Yaskawa INFORM job: A_ROOF_SIDE_0617_2_PAINT_52.JBI

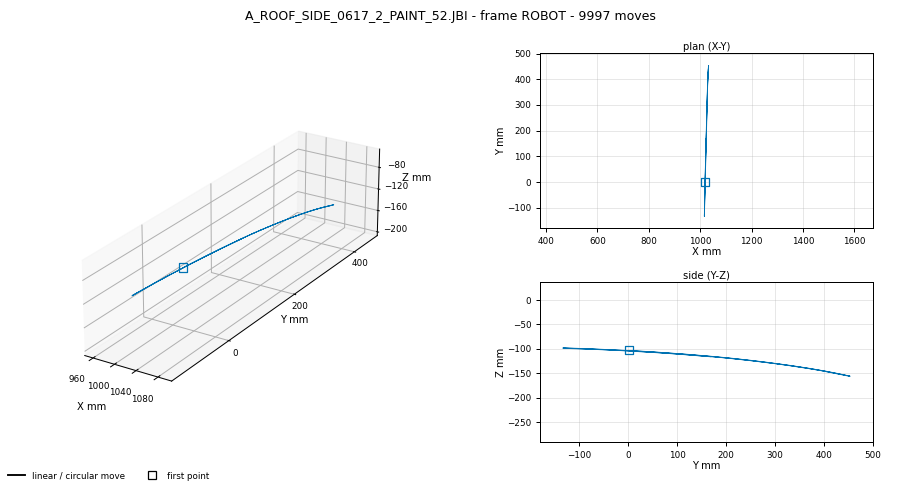
[picture p0: tool path of A_ROOF_SIDE_0617_2_PAINT_52.JBI in frame ROBOT, 9997 of 9997 moves have a stored position in this frame; points joined in program order, loops and branches not executed]
/JOB
//NAME A_ROOF_SIDE_0617_2_PAINT52
//POS
///NPOS 9997,0,0,0,0,0
///TOOL 1
///USER 0
///POSTYPE ROBOT
///RECTAN
///RCONF 1,0,0,0,0,0,0,0,0,0,0,0,0,0,0,0,0,0,0,0,0,0,0,0
C00000=1019.781,0.856,-102.921,166.512,52.317,159.512
C00001=1019.787,1.106,-102.935,166.515,52.311,159.512
C00002=1019.792,1.356,-102.949,166.518,52.306,159.511
C00003=1019.798,1.605,-102.963,166.520,52.301,159.511
C00004=1019.804,1.854,-102.976,166.523,52.295,159.510
C00005=1019.809,2.104,-102.990,166.526,52.289,159.510
C00006=1019.815,2.354,-103.004,166.529,52.284,159.509
C00007=1019.821,2.604,-103.018,166.531,52.279,159.509
C00008=1019.826,2.853,-103.032,166.533,52.273,159.508
C00009=1019.833,3.103,-103.045,166.536,52.268,159.508
C00010=1019.838,3.352,-103.059,166.540,52.262,159.507
C00011=1019.843,3.602,-103.073,166.541,52.257,159.506
C00012=1019.849,3.851,-103.087,166.544,52.251,159.506
C00013=1019.855,4.100,-103.101,166.547,52.246,159.506
C00014=1019.860,4.350,-103.115,166.550,52.240,159.505
C00015=1019.866,4.599,-103.128,166.553,52.235,159.505
C00016=1019.872,4.849,-103.142,166.555,52.230,159.504
C00017=1019.877,5.098,-103.156,166.558,52.224,159.503
C00018=1019.883,5.349,-103.170,166.561,52.218,159.503
C00019=1019.889,5.598,-103.184,166.564,52.213,159.503
C00020=1019.895,5.848,-103.197,166.565,52.207,159.502
C00021=1019.901,6.097,-103.211,166.569,52.202,159.501
C00022=1019.906,6.347,-103.225,166.572,52.197,159.501
C00023=1019.912,6.596,-103.240,166.574,52.191,159.500
C00024=1019.917,6.845,-103.254,166.577,52.186,159.500
C00025=1019.923,7.095,-103.268,166.579,52.180,159.499
C00026=1019.930,7.345,-103.281,166.582,52.175,159.499
C00027=1019.935,7.594,-103.295,166.585,52.169,159.498
C00028=1019.941,7.844,-103.309,166.588,52.163,159.498
C00029=1019.946,8.093,-103.323,166.591,52.158,159.497
C00030=1019.952,8.342,-103.337,166.594,52.152,159.497
C00031=1019.958,8.593,-103.351,166.596,52.147,159.496
C00032=1019.964,8.842,-103.365,166.598,52.141,159.496
C00033=1019.970,9.092,-103.379,166.601,52.136,159.495
C00034=1019.975,9.341,-103.392,166.604,52.130,159.495
C00035=1019.981,9.590,-103.407,166.607,52.124,159.494
C00036=1019.987,9.840,-103.421,166.609,52.119,159.493
C00037=1019.992,10.090,-103.435,166.612,52.113,159.493
C00038=1019.999,10.339,-103.448,166.614,52.107,159.492
C00039=1020.005,10.622,-103.464,166.618,52.101,159.492
C00040=1020.011,10.903,-103.481,166.621,52.095,159.491
C00041=1020.019,11.186,-103.496,166.623,52.089,159.491
C00042=1020.025,11.469,-103.512,166.627,52.083,159.490
C00043=1020.031,11.718,-103.526,166.630,52.077,159.490
C00044=1020.036,11.967,-103.541,166.633,52.071,159.489
C00045=1020.042,12.217,-103.554,166.635,52.066,159.488
C00046=1020.048,12.467,-103.569,166.637,52.060,159.488
C00047=1020.054,12.716,-103.583,166.640,52.055,159.487
C00048=1020.060,12.965,-103.597,166.643,52.049,159.487
C00049=1020.065,13.215,-103.610,166.646,52.043,159.486
C00050=1020.071,13.465,-103.625,166.649,52.037,159.486
C00051=1020.077,13.714,-103.639,166.651,52.032,159.485
C00052=1020.083,13.964,-103.653,166.654,52.026,159.485
C00053=1020.089,14.213,-103.668,166.657,52.021,159.484
C00054=1020.094,14.463,-103.682,166.660,52.016,159.484
C00055=1020.100,14.712,-103.697,166.661,52.010,159.483
C00056=1020.105,14.962,-103.711,166.664,52.005,159.483
C00057=1020.111,15.211,-103.726,166.667,51.999,159.482
C00058=1020.117,15.461,-103.740,166.670,51.994,159.482
C00059=1020.123,15.710,-103.754,166.672,51.989,159.481
C00060=1020.129,15.960,-103.769,166.675,51.983,159.480
C00061=1020.135,16.209,-103.783,166.678,51.977,159.480
C00062=1020.139,16.459,-103.798,166.681,51.971,159.479
C00063=1020.145,16.708,-103.812,166.683,51.966,159.479
C00064=1020.151,16.958,-103.826,166.685,51.960,159.478
C00065=1020.157,17.207,-103.841,166.689,51.955,159.478
C00066=1020.162,17.457,-103.855,166.691,51.949,159.477
C00067=1020.169,17.706,-103.870,166.693,51.944,159.477
C00068=1020.174,17.956,-103.884,166.696,51.938,159.476
C00069=1020.180,18.205,-103.898,166.699,51.933,159.476
C00070=1020.185,18.455,-103.913,166.702,51.927,159.475
C00071=1020.191,18.704,-103.928,166.705,51.922,159.475
C00072=1020.197,18.954,-103.941,166.707,51.916,159.474
C00073=1020.203,19.204,-103.956,166.710,51.911,159.473
C00074=1020.209,19.453,-103.971,166.713,51.906,159.473
C00075=1020.214,19.703,-103.986,166.715,51.900,159.472
C00076=1020.220,19.952,-104.000,166.717,51.895,159.472
C00077=1020.226,20.201,-104.015,166.720,51.889,159.471
C00078=1020.232,20.451,-104.029,166.723,51.883,159.471
C00079=1020.237,20.701,-104.044,166.725,51.878,159.470
C00080=1020.243,20.950,-104.059,166.728,51.873,159.470
C00081=1020.249,21.200,-104.073,166.731,51.867,159.469
C00082=1020.254,21.449,-104.088,166.734,51.861,159.469
C00083=1020.259,21.698,-104.103,166.736,51.856,159.468
C00084=1020.266,21.948,-104.117,166.739,51.850,159.467
C00085=1020.271,22.197,-104.132,166.741,51.844,159.467
C00086=1020.277,22.447,-104.147,166.744,51.839,159.466
C00087=1020.282,22.697,-104.161,166.746,51.834,159.466
C00088=1020.288,22.946,-104.176,166.749,51.828,159.465
C00089=1020.294,23.196,-104.191,166.752,51.822,159.465
C00090=1020.300,23.445,-104.206,166.755,51.817,159.464
C00091=1020.306,23.695,-104.220,166.758,51.811,159.463
C00092=1020.312,23.944,-104.235,166.760,51.806,159.463
C00093=1020.317,24.194,-104.250,166.762,51.800,159.462
C00094=1020.323,24.443,-104.265,166.766,51.795,159.462
C00095=1020.328,24.692,-104.279,166.768,51.789,159.461
C00096=1020.334,24.942,-104.294,166.770,51.784,159.461
C00097=1020.340,25.191,-104.309,166.773,51.778,159.460
C00098=1020.346,25.441,-104.324,166.776,51.773,159.460
C00099=1020.351,25.690,-104.339,166.779,51.767,159.459
C00100=1020.357,25.941,-104.353,166.781,51.761,159.458
C00101=1020.363,26.190,-104.368,166.784,51.756,159.458
C00102=1020.369,26.440,-104.383,166.786,51.750,159.457
C00103=1020.376,26.723,-104.400,166.789,51.744,159.457
C00104=1020.382,27.007,-104.417,166.793,51.738,159.456
C00105=1020.389,27.291,-104.434,166.795,51.731,159.455
C00106=1020.395,27.574,-104.450,166.799,51.725,159.455
C00107=1020.401,27.824,-104.465,166.801,51.719,159.454
C00108=1020.406,28.073,-104.481,166.804,51.714,159.454
C00109=1020.413,28.323,-104.496,166.807,51.709,159.453
C00110=1020.418,28.572,-104.511,166.809,51.703,159.452
C00111=1020.423,28.822,-104.526,166.812,51.698,159.452
C00112=1020.429,29.071,-104.541,166.814,51.692,159.451
C00113=1020.435,29.321,-104.556,166.817,51.687,159.451
C00114=1020.441,29.570,-104.571,166.819,51.681,159.450
C00115=1020.446,29.820,-104.586,166.822,51.676,159.450
C00116=1020.452,30.069,-104.601,166.825,51.670,159.449
C00117=1020.458,30.319,-104.617,166.828,51.664,159.449
C00118=1020.463,30.568,-104.631,166.830,51.659,159.448
C00119=1020.469,30.818,-104.647,166.833,51.653,159.447
C00120=1020.475,31.067,-104.661,166.836,51.648,159.447
C00121=1020.481,31.317,-104.677,166.837,51.642,159.446
C00122=1020.486,31.566,-104.691,166.840,51.637,159.446
C00123=1020.492,31.816,-104.707,166.843,51.631,159.445
C00124=1020.497,32.065,-104.722,166.846,51.626,159.445
C00125=1020.503,32.315,-104.737,166.848,51.620,159.444
C00126=1020.508,32.564,-104.752,166.851,51.614,159.443
C00127=1020.515,32.813,-104.768,166.854,51.609,159.443
C00128=1020.521,33.063,-104.783,166.857,51.603,159.442
C00129=1020.527,33.312,-104.798,166.859,51.598,159.442
C00130=1020.532,33.562,-104.814,166.861,51.592,159.441
C00131=1020.538,33.811,-104.828,166.864,51.586,159.441
C00132=1020.544,34.061,-104.844,166.867,51.581,159.440
C00133=1020.549,34.310,-104.858,166.869,51.576,159.439
C00134=1020.555,34.560,-104.874,166.872,51.570,159.439
C00135=1020.561,34.810,-104.889,166.875,51.564,159.438
C00136=1020.566,35.059,-104.904,166.878,51.559,159.438
C00137=1020.572,35.308,-104.920,166.880,51.554,159.437
C00138=1020.578,35.557,-104.935,166.882,51.548,159.437
C00139=1020.584,35.807,-104.950,166.885,51.542,159.436
C00140=1020.590,36.057,-104.965,166.888,51.537,159.435
C00141=1020.595,36.306,-104.980,166.891,51.531,159.435
C00142=1020.602,36.555,-104.995,166.893,51.525,159.434
C00143=1020.608,36.805,-105.012,166.896,51.520,159.434
C00144=1020.613,37.054,-105.027,166.899,51.514,159.433
C00145=1020.618,37.304,-105.042,166.901,51.509,159.432
C00146=1020.624,37.554,-105.058,166.903,51.503,159.432
C00147=1020.630,37.802,-105.073,166.907,51.498,159.431
C00148=1020.636,38.052,-105.089,166.909,51.492,159.431
C00149=1020.641,38.302,-105.104,166.911,51.486,159.430
C00150=1020.647,38.551,-105.120,166.914,51.481,159.430
C00151=1020.652,38.801,-105.136,166.917,51.475,159.429
C00152=1020.658,39.050,-105.150,166.919,51.470,159.428
C00153=1020.664,39.299,-105.167,166.922,51.464,159.428
C00154=1020.670,39.549,-105.182,166.925,51.459,159.427
C00155=1020.675,39.798,-105.197,166.928,51.453,159.427
C00156=1020.681,40.048,-105.214,166.929,51.448,159.426
C00157=1020.687,40.297,-105.228,166.932,51.443,159.426
C00158=1020.692,40.547,-105.244,166.935,51.437,159.425
C00159=1020.698,40.796,-105.260,166.937,51.432,159.424
C00160=1020.704,41.046,-105.275,166.940,51.426,159.424
C00161=1020.709,41.295,-105.291,166.943,51.420,159.423
C00162=1020.715,41.544,-105.306,166.946,51.415,159.423
C00163=1020.721,41.794,-105.322,166.948,51.409,159.422
C00164=1020.726,42.043,-105.338,166.950,51.403,159.421
C00165=1020.732,42.293,-105.353,166.954,51.398,159.421
C00166=1020.738,42.542,-105.369,166.955,51.392,159.420
C00167=1020.744,42.826,-105.386,166.959,51.386,159.420
C00168=1020.750,43.110,-105.405,166.962,51.380,159.419
C00169=1020.757,43.394,-105.423,166.965,51.374,159.418
C00170=1020.763,43.677,-105.441,166.968,51.367,159.418
C00171=1020.769,43.926,-105.457,166.970,51.363,159.417
C00172=1020.775,44.176,-105.473,166.973,51.357,159.417
C00173=1020.780,44.425,-105.489,166.976,51.351,159.416
C00174=1020.785,44.675,-105.505,166.978,51.346,159.415
C00175=1020.791,44.925,-105.521,166.981,51.341,159.415
C00176=1020.797,45.173,-105.537,166.984,51.335,159.414
C00177=1020.802,45.423,-105.552,166.986,51.330,159.414
C00178=1020.808,45.672,-105.569,166.989,51.324,159.413
C00179=1020.814,45.922,-105.584,166.992,51.319,159.413
C00180=1020.819,46.171,-105.600,166.993,51.313,159.412
C00181=1020.825,46.420,-105.616,166.997,51.308,159.412
C00182=1020.831,46.670,-105.632,166.999,51.302,159.411
C00183=1020.837,46.920,-105.648,167.001,51.297,159.410
C00184=1020.841,47.169,-105.665,167.004,51.291,159.410
C00185=1020.847,47.419,-105.680,167.007,51.285,159.409
C00186=1020.853,47.668,-105.697,167.009,51.281,159.409
C00187=1020.859,47.917,-105.713,167.012,51.275,159.408
C00188=1020.864,48.167,-105.728,167.015,51.269,159.407
C00189=1020.870,48.416,-105.744,167.017,51.264,159.407
C00190=1020.876,48.665,-105.760,167.020,51.258,159.406
C00191=1020.881,48.915,-105.776,167.023,51.253,159.406
C00192=1020.887,49.165,-105.792,167.024,51.247,159.405
C00193=1020.893,49.413,-105.808,167.027,51.241,159.404
C00194=1020.898,49.663,-105.825,167.030,51.236,159.404
C00195=1020.904,49.913,-105.841,167.032,51.231,159.403
C00196=1020.910,50.162,-105.857,167.035,51.226,159.403
C00197=1020.916,50.412,-105.873,167.038,51.220,159.402
C00198=1020.921,50.661,-105.888,167.041,51.214,159.401
C00199=1020.927,50.910,-105.904,167.043,51.209,159.401
C00200=1020.932,51.160,-105.921,167.046,51.203,159.400
C00201=1020.938,51.409,-105.937,167.049,51.197,159.400
C00202=1020.944,51.659,-105.953,167.051,51.192,159.399
C00203=1020.950,51.908,-105.969,167.053,51.186,159.398
C00204=1020.955,52.157,-105.985,167.056,51.181,159.398
C00205=1020.961,52.407,-106.002,167.059,51.175,159.397
C00206=1020.967,52.656,-106.018,167.061,51.170,159.397
C00207=1020.972,52.906,-106.033,167.064,51.164,159.396
C00208=1020.978,53.155,-106.050,167.067,51.158,159.395
C00209=1020.984,53.405,-106.066,167.070,51.153,159.395
C00210=1020.990,53.654,-106.082,167.072,51.147,159.394
C00211=1020.995,53.903,-106.098,167.074,51.141,159.394
C00212=1021.000,54.153,-106.114,167.077,51.136,159.393
C00213=1021.006,54.402,-106.130,167.079,51.131,159.392
C00214=1021.012,54.652,-106.147,167.082,51.125,159.392
C00215=1021.018,54.901,-106.163,167.085,51.119,159.391
C00216=1021.024,55.150,-106.179,167.088,51.113,159.390
C00217=1021.030,55.400,-106.195,167.090,51.108,159.390
C00218=1021.036,55.650,-106.211,167.093,51.102,159.389
C00219=1021.042,55.899,-106.227,167.095,51.096,159.389
C00220=1021.047,56.148,-106.243,167.098,51.091,159.388
C00221=1021.052,56.397,-106.260,167.100,51.086,159.387
C00222=1021.058,56.647,-106.276,167.103,51.080,159.387
C00223=1021.064,56.896,-106.292,167.106,51.074,159.386
C00224=1021.070,57.145,-106.309,167.109,51.068,159.386
C00225=1021.076,57.395,-106.325,167.112,51.062,159.385
C00226=1021.082,57.644,-106.341,167.114,51.057,159.384
C00227=1021.088,57.894,-106.357,167.116,51.052,159.384
C00228=1021.094,58.143,-106.373,167.119,51.046,159.383
C00229=1021.099,58.393,-106.390,167.122,51.040,159.382
C00230=1021.105,58.642,-106.406,167.124,51.034,159.382
C00231=1021.112,58.925,-106.425,167.128,51.028,159.381
C00232=1021.118,59.209,-106.443,167.130,51.022,159.380
C00233=1021.124,59.493,-106.461,167.133,51.015,159.380
C00234=1021.132,59.776,-106.480,167.136,51.009,159.379
C00235=1021.138,60.025,-106.496,167.139,51.003,159.378
C00236=1021.143,60.275,-106.513,167.142,50.997,159.378
C00237=1021.149,60.524,-106.530,167.145,50.991,159.377
C00238=1021.155,60.773,-106.546,167.146,50.986,159.376
C00239=1021.161,61.023,-106.562,167.149,50.980,159.376
C00240=1021.167,61.272,-106.578,167.152,50.975,159.375
C00241=1021.173,61.522,-106.595,167.155,50.969,159.375
C00242=1021.179,61.771,-106.611,167.158,50.963,159.374
C00243=1021.184,62.021,-106.628,167.160,50.957,159.373
C00244=1021.190,62.270,-106.644,167.163,50.952,159.373
C00245=1021.196,62.519,-106.660,167.165,50.946,159.372
C00246=1021.202,62.769,-106.676,167.168,50.940,159.371
C00247=1021.208,63.018,-106.693,167.171,50.934,159.371
C00248=1021.213,63.268,-106.710,167.173,50.929,159.370
C00249=1021.219,63.517,-106.726,167.176,50.923,159.370
C00250=1021.224,63.767,-106.743,167.179,50.918,159.369
C00251=1021.230,64.016,-106.759,167.181,50.912,159.368
C00252=1021.236,64.265,-106.776,167.183,50.906,159.368
C00253=1021.241,64.514,-106.793,167.187,50.901,159.367
C00254=1021.247,64.764,-106.809,167.189,50.895,159.366
C00255=1021.252,65.013,-106.826,167.191,50.890,159.366
C00256=1021.258,65.263,-106.842,167.194,50.884,159.365
C00257=1021.265,65.512,-106.860,167.197,50.879,159.365
C00258=1021.271,65.762,-106.876,167.200,50.873,159.364
C00259=1021.276,66.011,-106.893,167.202,50.867,159.363
C00260=1021.282,66.261,-106.909,167.205,50.862,159.363
C00261=1021.287,66.510,-106.927,167.208,50.856,159.362
C00262=1021.293,66.759,-106.943,167.210,50.851,159.361
C00263=1021.298,67.009,-106.960,167.212,50.845,159.361
C00264=1021.304,67.258,-106.976,167.215,50.839,159.360
C00265=1021.310,67.507,-106.994,167.218,50.833,159.360
C00266=1021.316,67.757,-107.010,167.220,50.829,159.359
C00267=1021.321,68.006,-107.027,167.223,50.823,159.358
C00268=1021.327,68.255,-107.044,167.226,50.817,159.358
C00269=1021.332,68.505,-107.061,167.229,50.811,159.357
C00270=1021.338,68.754,-107.077,167.231,50.806,159.357
C00271=1021.345,69.004,-107.095,167.234,50.800,159.356
C00272=1021.350,69.253,-107.112,167.237,50.795,159.355
C00273=1021.356,69.502,-107.129,167.238,50.789,159.354
C00274=1021.361,69.752,-107.146,167.242,50.784,159.354
C00275=1021.367,70.001,-107.162,167.244,50.778,159.353
C00276=1021.373,70.250,-107.179,167.247,50.772,159.353
C00277=1021.378,70.500,-107.196,167.249,50.767,159.352
C00278=1021.384,70.749,-107.213,167.252,50.762,159.352
C00279=1021.389,70.998,-107.230,167.255,50.756,159.351
C00280=1021.395,71.247,-107.248,167.257,50.750,159.350
C00281=1021.401,71.497,-107.264,167.260,50.744,159.350
C00282=1021.407,71.747,-107.281,167.263,50.739,159.349
C00283=1021.412,71.996,-107.299,167.266,50.734,159.348
C00284=1021.418,72.245,-107.315,167.268,50.728,159.348
C00285=1021.424,72.494,-107.333,167.270,50.722,159.347
C00286=1021.429,72.744,-107.349,167.274,50.717,159.347
C00287=1021.435,72.993,-107.366,167.275,50.712,159.346
C00288=1021.440,73.242,-107.383,167.278,50.706,159.345
C00289=1021.446,73.492,-107.401,167.281,50.700,159.345
C00290=1021.452,73.742,-107.417,167.284,50.694,159.344
C00291=1021.458,73.991,-107.435,167.286,50.689,159.343
C00292=1021.463,74.240,-107.452,167.289,50.684,159.343
C00293=1021.469,74.489,-107.469,167.292,50.678,159.342
C00294=1021.475,74.738,-107.486,167.295,50.672,159.342
C00295=1021.482,75.022,-107.506,167.297,50.666,159.341
C00296=1021.488,75.305,-107.526,167.300,50.660,159.340
C00297=1021.495,75.589,-107.545,167.303,50.653,159.339
C00298=1021.501,75.872,-107.564,167.306,50.647,159.339
C00299=1021.507,76.122,-107.582,167.309,50.641,159.338
C00300=1021.512,76.371,-107.599,167.312,50.635,159.337
C00301=1021.518,76.620,-107.616,167.314,50.630,159.337
C00302=1021.524,76.870,-107.633,167.317,50.624,159.336
C00303=1021.529,77.119,-107.650,167.320,50.619,159.336
C00304=1021.535,77.368,-107.668,167.323,50.613,159.335
C00305=1021.540,77.618,-107.685,167.324,50.608,159.334
C00306=1021.546,77.867,-107.703,167.327,50.602,159.334
C00307=1021.551,78.116,-107.720,167.331,50.597,159.333
C00308=1021.558,78.366,-107.738,167.332,50.591,159.332
C00309=1021.563,78.616,-107.755,167.335,50.585,159.332
C00310=1021.568,78.865,-107.772,167.338,50.580,159.331
C00311=1021.574,79.114,-107.790,167.340,50.575,159.331
C00312=1021.579,79.363,-107.808,167.343,50.569,159.330
C00313=1021.585,79.613,-107.825,167.346,50.563,159.329
C00314=1021.591,79.862,-107.842,167.349,50.558,159.329
C00315=1021.596,80.111,-107.860,167.351,50.553,159.328
C00316=1021.602,80.360,-107.877,167.354,50.547,159.327
C00317=1021.608,80.610,-107.895,167.357,50.541,159.327
C00318=1021.613,80.860,-107.912,167.359,50.536,159.326
C00319=1021.619,81.109,-107.930,167.362,50.530,159.326
C00320=1021.625,81.357,-107.947,167.365,50.525,159.325
C00321=1021.631,81.607,-107.965,167.367,50.519,159.324
C00322=1021.637,81.856,-107.982,167.370,50.514,159.324
C00323=1021.642,82.105,-108.000,167.373,50.508,159.323
C00324=1021.647,82.355,-108.017,167.375,50.503,159.323
C00325=1021.653,82.605,-108.035,167.377,50.497,159.322
C00326=1021.659,82.854,-108.052,167.380,50.491,159.321
C00327=1021.664,83.103,-108.070,167.383,50.486,159.321
C00328=1021.670,83.352,-108.087,167.386,50.480,159.320
C00329=1021.676,83.601,-108.105,167.388,50.475,159.319
C00330=1021.682,83.850,-108.123,167.391,50.469,159.319
C00331=1021.687,84.099,-108.140,167.394,50.463,159.318
C00332=1021.693,84.350,-108.158,167.397,50.458,159.318
C00333=1021.698,84.599,-108.175,167.399,50.453,159.317
C00334=1021.704,84.848,-108.193,167.402,50.447,159.316
C00335=1021.710,85.098,-108.211,167.405,50.441,159.316
C00336=1021.716,85.347,-108.228,167.407,50.435,159.315
C00337=1021.721,85.596,-108.246,167.409,50.430,159.314
C00338=1021.727,85.845,-108.264,167.412,50.424,159.314
C00339=1021.733,86.095,-108.281,167.415,50.419,159.313
C00340=1021.738,86.344,-108.299,167.418,50.413,159.312
C00341=1021.744,86.593,-108.317,167.420,50.408,159.312
C00342=1021.750,86.842,-108.334,167.423,50.402,159.311
C00343=1021.755,87.091,-108.352,167.426,50.396,159.310
C00344=1021.762,87.341,-108.370,167.429,50.391,159.310
C00345=1021.767,87.590,-108.387,167.432,50.385,159.309
C00346=1021.773,87.839,-108.405,167.433,50.379,159.308
C00347=1021.779,88.089,-108.423,167.437,50.374,159.308
C00348=1021.784,88.338,-108.441,167.440,50.368,159.307
C00349=1021.790,88.588,-108.458,167.442,50.363,159.307
C00350=1021.796,88.837,-108.476,167.445,50.357,159.306
C00351=1021.801,89.086,-108.494,167.447,50.351,159.305
C00352=1021.807,89.336,-108.512,167.450,50.346,159.305
C00353=1021.812,89.585,-108.530,167.453,50.340,159.304
C00354=1021.818,89.835,-108.548,167.456,50.335,159.304
C00355=1021.824,90.084,-108.565,167.458,50.329,159.303
C00356=1021.829,90.333,-108.583,167.461,50.324,159.302
C00357=1021.835,90.583,-108.601,167.464,50.318,159.302
C00358=1021.841,90.831,-108.620,167.466,50.313,159.301
C00359=1021.847,91.115,-108.640,167.470,50.306,159.300
C00360=1021.853,91.398,-108.660,167.472,50.301,159.300
C00361=1021.859,91.682,-108.681,167.475,50.294,159.299
C00362=1021.866,91.965,-108.701,167.479,50.288,159.298
C00363=1021.874,92.347,-108.729,167.483,50.280,159.297
C00364=1021.883,92.730,-108.757,167.486,50.271,159.296
C00365=1021.892,93.111,-108.784,167.491,50.262,159.295
C00366=1021.900,93.494,-108.812,167.495,50.254,159.294
C00367=1021.906,93.743,-108.830,167.498,50.248,159.294
C00368=1021.911,93.992,-108.848,167.500,50.243,159.293
C00369=1021.917,94.242,-108.866,167.503,50.238,159.292
C00370=1021.923,94.491,-108.884,167.506,50.232,159.292
C00371=1021.929,94.740,-108.903,167.509,50.226,159.291
C00372=1021.934,94.989,-108.921,167.511,50.221,159.290
C00373=1021.940,95.239,-108.939,167.514,50.215,159.290
C00374=1021.945,95.488,-108.958,167.517,50.210,159.289
C00375=1021.951,95.737,-108.975,167.520,50.204,159.289
C00376=1021.957,95.987,-108.993,167.522,50.199,159.288
C00377=1021.962,96.235,-109.012,167.525,50.193,159.287
C00378=1021.968,96.485,-109.030,167.528,50.187,159.287
C00379=1021.974,96.734,-109.047,167.530,50.181,159.286
C00380=1021.980,96.983,-109.066,167.533,50.176,159.285
C00381=1021.985,97.233,-109.084,167.536,50.171,159.285
C00382=1021.991,97.482,-109.102,167.538,50.165,159.284
C00383=1021.997,97.731,-109.120,167.541,50.159,159.284
C00384=1022.002,97.981,-109.139,167.544,50.154,159.283
C00385=1022.008,98.230,-109.157,167.547,50.148,159.282
C00386=1022.014,98.479,-109.175,167.549,50.142,159.281
C00387=1022.019,98.728,-109.193,167.552,50.137,159.281
C00388=1022.025,98.978,-109.211,167.555,50.131,159.280
C00389=1022.031,99.227,-109.230,167.558,50.126,159.280
C00390=1022.036,99.477,-109.248,167.561,50.120,159.279
C00391=1022.042,99.725,-109.266,167.563,50.115,159.278
C00392=1022.047,99.975,-109.285,167.566,50.109,159.278
C00393=1022.052,100.224,-109.304,167.569,50.104,159.277
C00394=1022.059,100.474,-109.322,167.571,50.099,159.277
C00395=1022.064,100.723,-109.341,167.574,50.093,159.276
C00396=1022.070,100.972,-109.359,167.577,50.087,159.275
C00397=1022.075,101.221,-109.378,167.580,50.082,159.275
C00398=1022.081,101.470,-109.397,167.582,50.077,159.274
C00399=1022.087,101.720,-109.415,167.585,50.071,159.273
C00400=1022.092,101.969,-109.433,167.588,50.065,159.273
C00401=1022.098,102.218,-109.451,167.591,50.060,159.272
C00402=1022.103,102.467,-109.470,167.593,50.055,159.272
C00403=1022.109,102.717,-109.490,167.596,50.049,159.271
C00404=1022.114,102.966,-109.507,167.599,50.043,159.270
C00405=1022.120,103.215,-109.526,167.602,50.038,159.270
C00406=1022.125,103.464,-109.544,167.604,50.033,159.269
C00407=1022.131,103.713,-109.563,167.607,50.027,159.268
C00408=1022.137,103.963,-109.582,167.610,50.021,159.268
C00409=1022.142,104.212,-109.600,167.613,50.016,159.267
C00410=1022.148,104.461,-109.619,167.616,50.011,159.267
C00411=1022.154,104.710,-109.637,167.618,50.005,159.266
C00412=1022.159,104.960,-109.656,167.621,49.999,159.265
C00413=1022.165,105.209,-109.675,167.624,49.994,159.265
C00414=1022.171,105.458,-109.694,167.627,49.988,159.264
C00415=1022.176,105.708,-109.712,167.629,49.983,159.263
C00416=1022.181,105.956,-109.731,167.632,49.978,159.263
C00417=1022.188,106.206,-109.750,167.635,49.972,159.262
C00418=1022.193,106.456,-109.768,167.638,49.966,159.262
C00419=1022.203,106.855,-109.798,167.643,49.957,159.261
C00420=1022.211,107.255,-109.828,167.646,49.948,159.259
C00421=1022.220,107.655,-109.858,167.651,49.940,159.258
C00422=1022.229,108.055,-109.887,167.656,49.931,159.258
C00423=1022.235,108.305,-109.907,167.659,49.925,159.257
C00424=1022.240,108.553,-109.926,167.661,49.920,159.256
C00425=1022.247,108.802,-109.944,167.664,49.914,159.256
C00426=1022.252,109.052,-109.963,167.667,49.908,159.255
C00427=1022.257,109.301,-109.982,167.670,49.903,159.254
C00428=1022.264,109.550,-110.000,167.672,49.897,159.254
C00429=1022.269,109.800,-110.019,167.675,49.892,159.253
C00430=1022.274,110.048,-110.038,167.678,49.886,159.252
C00431=1022.280,110.298,-110.057,167.681,49.881,159.252
C00432=1022.286,110.548,-110.076,167.684,49.875,159.251
C00433=1022.291,110.796,-110.094,167.686,49.869,159.250
C00434=1022.297,111.046,-110.114,167.689,49.865,159.250
C00435=1022.303,111.295,-110.133,167.692,49.859,159.249
C00436=1022.308,111.544,-110.152,167.695,49.853,159.249
C00437=1022.314,111.793,-110.170,167.698,49.848,159.248
C00438=1022.320,112.042,-110.190,167.701,49.842,159.247
C00439=1022.326,112.292,-110.209,167.703,49.837,159.247
C00440=1022.331,112.541,-110.228,167.706,49.831,159.246
C00441=1022.336,112.790,-110.247,167.709,49.826,159.245
C00442=1022.342,113.040,-110.266,167.712,49.821,159.245
C00443=1022.347,113.288,-110.285,167.714,49.815,159.244
C00444=1022.353,113.538,-110.304,167.717,49.810,159.244
C00445=1022.358,113.787,-110.324,167.720,49.805,159.243
C00446=1022.364,114.036,-110.343,167.723,49.799,159.243
C00447=1022.369,114.285,-110.362,167.725,49.794,159.242
C00448=1022.374,114.535,-110.382,167.728,49.789,159.241
C00449=1022.380,114.784,-110.401,167.731,49.783,159.241
C00450=1022.385,115.033,-110.420,167.734,49.777,159.240
C00451=1022.391,115.283,-110.439,167.736,49.772,159.239
C00452=1022.396,115.532,-110.458,167.739,49.767,159.239
C00453=1022.402,115.780,-110.478,167.742,49.761,159.238
C00454=1022.407,116.030,-110.497,167.746,49.756,159.238
C00455=1022.413,116.279,-110.516,167.749,49.750,159.237
C00456=1022.419,116.528,-110.536,167.751,49.745,159.236
C00457=1022.424,116.777,-110.554,167.754,49.739,159.236
C00458=1022.429,117.027,-110.574,167.757,49.734,159.235
C00459=1022.435,117.276,-110.594,167.760,49.729,159.235
C00460=1022.440,117.525,-110.613,167.762,49.723,159.234
C00461=1022.446,117.774,-110.632,167.765,49.718,159.233
C00462=1022.451,118.023,-110.652,167.768,49.713,159.233
C00463=1022.457,118.273,-110.671,167.771,49.707,159.232
C00464=1022.463,118.522,-110.690,167.774,49.702,159.232
C00465=1022.469,118.771,-110.710,167.776,49.697,159.231
C00466=1022.474,119.020,-110.729,167.779,49.691,159.230
C00467=1022.479,119.269,-110.748,167.782,49.685,159.230
C00468=1022.484,119.519,-110.768,167.785,49.680,159.229
C00469=1022.490,119.768,-110.788,167.788,49.675,159.228
C00470=1022.495,120.016,-110.807,167.791,49.669,159.228
C00471=1022.501,120.266,-110.826,167.793,49.664,159.227
C00472=1022.507,120.515,-110.845,167.797,49.659,159.227
C00473=1022.513,120.764,-110.865,167.800,49.653,159.226
C00474=1022.518,121.014,-110.885,167.803,49.647,159.225
C00475=1022.524,121.263,-110.904,167.805,49.642,159.225
C00476=1022.529,121.512,-110.923,167.809,49.637,159.224
C00477=1022.535,121.761,-110.943,167.811,49.631,159.223
C00478=1022.540,122.010,-110.962,167.814,49.625,159.223
C00479=1022.546,122.260,-110.982,167.817,49.620,159.222
C00480=1022.552,122.509,-111.002,167.820,49.615,159.222
C00481=1022.558,122.758,-111.021,167.823,49.609,159.221
C00482=1022.563,123.007,-111.040,167.826,49.604,159.220
C00483=1022.569,123.290,-111.062,167.829,49.598,159.220
C00484=1022.576,123.574,-111.084,167.833,49.591,159.219
C00485=1022.582,123.858,-111.107,167.835,49.585,159.218
C00486=1022.588,124.141,-111.129,167.839,49.579,159.218
C00487=1022.594,124.390,-111.148,167.842,49.573,159.217
C00488=1022.600,124.639,-111.168,167.845,49.568,159.216
C00489=1022.606,124.888,-111.187,167.847,49.562,159.216
C00490=1022.611,125.137,-111.208,167.850,49.557,159.215
C00491=1022.617,125.387,-111.227,167.853,49.552,159.214
C00492=1022.622,125.636,-111.246,167.856,49.546,159.214
C00493=1022.628,125.885,-111.266,167.859,49.540,159.213
C00494=1022.634,126.135,-111.285,167.862,49.535,159.213
C00495=1022.640,126.383,-111.305,167.866,49.530,159.212
C00496=1022.645,126.632,-111.324,167.869,49.524,159.211
C00497=1022.651,126.881,-111.343,167.872,49.518,159.211
C00498=1022.656,127.131,-111.364,167.875,49.513,159.210
C00499=1022.662,127.380,-111.383,167.876,49.507,159.209
C00500=1022.668,127.629,-111.403,167.880,49.502,159.209
C00501=1022.673,127.878,-111.422,167.883,49.497,159.208
C00502=1022.679,128.127,-111.442,167.886,49.491,159.208
C00503=1022.685,128.377,-111.462,167.889,49.485,159.207
C00504=1022.691,128.625,-111.482,167.892,49.480,159.206
C00505=1022.696,128.875,-111.501,167.895,49.474,159.206
C00506=1022.702,129.124,-111.521,167.898,49.469,159.205
C00507=1022.708,129.373,-111.541,167.901,49.463,159.205
C00508=1022.714,129.622,-111.561,167.904,49.458,159.204
C00509=1022.719,129.872,-111.580,167.907,49.452,159.203
C00510=1022.725,130.120,-111.600,167.910,49.447,159.203
C00511=1022.730,130.370,-111.620,167.913,49.442,159.202
C00512=1022.736,130.619,-111.640,167.915,49.436,159.201
C00513=1022.742,130.868,-111.660,167.918,49.431,159.201
C00514=1022.747,131.118,-111.679,167.922,49.426,159.200
C00515=1022.752,131.367,-111.700,167.925,49.420,159.200
C00516=1022.758,131.615,-111.720,167.928,49.414,159.199
C00517=1022.763,131.865,-111.740,167.931,49.409,159.199
C00518=1022.769,132.114,-111.760,167.934,49.404,159.198
C00519=1022.775,132.363,-111.780,167.936,49.398,159.197
C00520=1022.781,132.612,-111.800,167.939,49.393,159.197
C00521=1022.786,132.862,-111.820,167.942,49.388,159.196
C00522=1022.792,133.111,-111.840,167.945,49.382,159.195
C00523=1022.797,133.360,-111.861,167.948,49.377,159.195
C00524=1022.803,133.608,-111.881,167.952,49.372,159.194
C00525=1022.809,133.858,-111.900,167.955,49.366,159.194
C00526=1022.814,134.107,-111.920,167.958,49.360,159.193
C00527=1022.820,134.356,-111.940,167.961,49.355,159.192
C00528=1022.825,134.605,-111.961,167.964,49.350,159.192
C00529=1022.831,134.854,-111.980,167.966,49.344,159.191
C00530=1022.836,135.103,-112.001,167.969,49.340,159.191
C00531=1022.842,135.352,-112.021,167.972,49.334,159.190
C00532=1022.847,135.601,-112.041,167.975,49.328,159.189
C00533=1022.853,135.850,-112.061,167.979,49.323,159.189
C00534=1022.858,136.100,-112.081,167.982,49.318,159.188
C00535=1022.864,136.349,-112.101,167.985,49.312,159.188
C00536=1022.869,136.598,-112.121,167.988,49.307,159.187
C00537=1022.875,136.847,-112.142,167.991,49.302,159.186
C00538=1022.881,137.097,-112.162,167.994,49.296,159.186
C00539=1022.887,137.346,-112.183,167.997,49.291,159.185
C00540=1022.893,137.595,-112.203,168.000,49.285,159.185
C00541=1022.898,137.844,-112.223,168.003,49.280,159.184
C00542=1022.904,138.092,-112.243,168.006,49.275,159.183
C00543=1022.909,138.342,-112.263,168.009,49.269,159.183
C00544=1022.914,138.591,-112.284,168.012,49.264,159.182
C00545=1022.919,138.840,-112.304,168.015,49.259,159.182
C00546=1022.925,139.089,-112.324,168.018,49.253,159.181
C00547=1022.931,139.373,-112.348,168.022,49.247,159.180
C00548=1022.937,139.656,-112.372,168.025,49.241,159.180
C00549=1022.944,139.939,-112.395,168.029,49.235,159.179
C00550=1022.950,140.222,-112.418,168.032,49.230,159.178
C00551=1022.956,140.471,-112.439,168.035,49.224,159.178
C00552=1022.962,140.721,-112.460,168.038,49.218,159.177
C00553=1022.968,140.970,-112.480,168.041,49.213,159.177
C00554=1022.973,141.219,-112.500,168.044,49.208,159.176
C00555=1022.978,141.468,-112.521,168.048,49.203,159.175
C00556=1022.983,141.717,-112.541,168.051,49.197,159.175
C00557=1022.989,141.966,-112.561,168.054,49.192,159.174
C00558=1022.995,142.215,-112.582,168.057,49.187,159.174
C00559=1023.000,142.465,-112.603,168.060,49.181,159.173
C00560=1023.006,142.714,-112.623,168.063,49.176,159.172
C00561=1023.012,142.963,-112.644,168.066,49.171,159.172
C00562=1023.017,143.212,-112.665,168.069,49.165,159.171
C00563=1023.022,143.461,-112.685,168.073,49.160,159.171
C00564=1023.028,143.710,-112.706,168.076,49.154,159.170
C00565=1023.034,143.959,-112.726,168.079,49.149,159.169
C00566=1023.040,144.209,-112.747,168.082,49.144,159.169
C00567=1023.045,144.458,-112.767,168.085,49.138,159.168
C00568=1023.050,144.706,-112.788,168.088,49.133,159.168
C00569=1023.056,144.955,-112.808,168.092,49.128,159.167
C00570=1023.062,145.205,-112.829,168.095,49.122,159.167
C00571=1023.068,145.454,-112.850,168.098,49.117,159.166
C00572=1023.073,145.703,-112.870,168.101,49.112,159.165
C00573=1023.079,145.951,-112.891,168.104,49.106,159.165
C00574=1023.085,146.201,-112.912,168.107,49.101,159.164
C00575=1023.090,146.450,-112.932,168.109,49.096,159.164
C00576=1023.095,146.699,-112.953,168.113,49.091,159.163
C00577=1023.101,146.948,-112.974,168.116,49.085,159.162
C00578=1023.106,147.197,-112.995,168.119,49.081,159.162
C00579=1023.112,147.447,-113.016,168.122,49.075,159.161
C00580=1023.118,147.695,-113.037,168.125,49.069,159.161
C00581=1023.123,147.944,-113.058,168.129,49.064,159.160
C00582=1023.128,148.193,-113.079,168.132,49.059,159.160
C00583=1023.134,148.443,-113.100,168.135,49.054,159.159
C00584=1023.140,148.692,-113.120,168.138,49.048,159.158
C00585=1023.145,148.940,-113.142,168.141,49.043,159.158
C00586=1023.151,149.190,-113.163,168.145,49.038,159.157
C00587=1023.157,149.439,-113.184,168.148,49.033,159.157
C00588=1023.162,149.688,-113.204,168.151,49.027,159.156
C00589=1023.167,149.937,-113.225,168.154,49.022,159.156
C00590=1023.173,150.186,-113.247,168.157,49.017,159.155
C00591=1023.179,150.435,-113.267,168.161,49.012,159.155
C00592=1023.184,150.684,-113.288,168.164,49.006,159.154
C00593=1023.190,150.934,-113.309,168.167,49.002,159.153
C00594=1023.195,151.182,-113.331,168.170,48.996,159.153
C00595=1023.201,151.431,-113.351,168.174,48.991,159.152
C00596=1023.206,151.680,-113.372,168.177,48.985,159.152
C00597=1023.212,151.930,-113.393,168.180,48.981,159.151
C00598=1023.218,152.178,-113.415,168.183,48.975,159.151
C00599=1023.223,152.427,-113.435,168.186,48.969,159.150
C00600=1023.229,152.676,-113.457,168.189,48.965,159.149
C00601=1023.234,152.925,-113.477,168.193,48.959,159.149
C00602=1023.239,153.174,-113.499,168.196,48.954,159.148
C00603=1023.245,153.424,-113.520,168.199,48.949,159.148
C00604=1023.251,153.673,-113.541,168.202,48.944,159.147
C00605=1023.257,153.922,-113.563,168.205,48.938,159.146
C00606=1023.262,154.171,-113.584,168.209,48.933,159.146
C00607=1023.268,154.419,-113.605,168.212,48.928,159.146
C00608=1023.273,154.669,-113.627,168.215,48.923,159.145
C00609=1023.278,154.918,-113.648,168.219,48.918,159.144
C00610=1023.284,155.167,-113.669,168.222,48.912,159.144
C00611=1023.290,155.450,-113.693,168.226,48.906,159.143
C00612=1023.297,155.733,-113.717,168.230,48.901,159.143
C00613=1023.303,156.016,-113.742,168.234,48.895,159.142
C00614=1023.310,156.299,-113.765,168.237,48.888,159.141
C00615=1023.314,156.548,-113.787,168.240,48.884,159.141
C00616=1023.321,156.797,-113.809,168.243,48.878,159.140
C00617=1023.326,157.046,-113.830,168.246,48.873,159.140
C00618=1023.332,157.296,-113.851,168.249,48.868,159.139
C00619=1023.338,157.544,-113.872,168.254,48.862,159.139
C00620=1023.342,157.793,-113.894,168.257,48.857,159.138
C00621=1023.348,158.042,-113.916,168.260,48.852,159.137
C00622=1023.354,158.291,-113.936,168.264,48.847,159.137
C00623=1023.360,158.541,-113.958,168.267,48.842,159.136
C00624=1023.365,158.789,-113.979,168.270,48.837,159.136
C00625=1023.371,159.039,-114.001,168.273,48.831,159.135
C00626=1023.376,159.287,-114.023,168.277,48.826,159.135
C00627=1023.381,159.537,-114.044,168.280,48.821,159.134
C00628=1023.386,159.786,-114.066,168.283,48.816,159.134
C00629=1023.392,160.035,-114.087,168.287,48.811,159.133
C00630=1023.398,160.284,-114.110,168.290,48.806,159.133
C00631=1023.403,160.532,-114.131,168.293,48.801,159.132
C00632=1023.409,160.782,-114.154,168.296,48.796,159.131
C00633=1023.414,161.030,-114.176,168.300,48.791,159.131
C00634=1023.419,161.279,-114.197,168.303,48.786,159.130
C00635=1023.424,161.528,-114.219,168.307,48.781,159.130
C00636=1023.429,161.777,-114.241,168.310,48.775,159.129
C00637=1023.435,162.026,-114.263,168.313,48.771,159.129
C00638=1023.440,162.275,-114.284,168.316,48.766,159.128
C00639=1023.446,162.525,-114.307,168.320,48.761,159.128
C00640=1023.451,162.773,-114.328,168.323,48.756,159.127
C00641=1023.457,163.023,-114.350,168.326,48.750,159.127
C00642=1023.462,163.272,-114.372,168.330,48.746,159.126
C00643=1023.468,163.521,-114.394,168.333,48.741,159.126
C00644=1023.473,163.770,-114.416,168.337,48.736,159.125
C00645=1023.478,164.018,-114.438,168.340,48.730,159.125
C00646=1023.484,164.267,-114.460,168.343,48.726,159.124
C00647=1023.489,164.516,-114.482,168.346,48.721,159.124
C00648=1023.494,164.765,-114.504,168.350,48.716,159.123
C00649=1023.500,165.015,-114.525,168.353,48.710,159.123
C00650=1023.505,165.263,-114.547,168.356,48.705,159.122
C00651=1023.511,165.512,-114.570,168.360,48.701,159.122
C00652=1023.516,165.761,-114.592,168.364,48.695,159.121
C00653=1023.522,166.010,-114.614,168.367,48.690,159.121
C00654=1023.527,166.259,-114.636,168.371,48.685,159.120
C00655=1023.533,166.508,-114.657,168.374,48.680,159.120
C00656=1023.538,166.756,-114.680,168.378,48.675,159.119
C00657=1023.543,167.006,-114.702,168.381,48.670,159.118
C00658=1023.549,167.254,-114.723,168.384,48.665,159.118
C00659=1023.554,167.504,-114.746,168.387,48.660,159.117
C00660=1023.560,167.753,-114.769,168.391,48.655,159.117
C00661=1023.566,168.001,-114.790,168.394,48.650,159.116
C00662=1023.571,168.251,-114.812,168.397,48.645,159.116
C00663=1023.576,168.500,-114.834,168.402,48.640,159.115
C00664=1023.582,168.748,-114.856,168.405,48.635,159.115
C00665=1023.588,168.998,-114.878,168.408,48.629,159.114
C00666=1023.593,169.247,-114.900,168.412,48.625,159.114
C00667=1023.599,169.495,-114.923,168.415,48.620,159.113
C00668=1023.604,169.745,-114.945,168.419,48.615,159.113
C00669=1023.609,169.994,-114.967,168.422,48.609,159.112
C00670=1023.616,170.242,-114.989,168.426,48.604,159.112
C00671=1023.621,170.491,-115.011,168.429,48.599,159.111
C00672=1023.626,170.740,-115.033,168.433,48.595,159.111
C00673=1023.632,170.989,-115.056,168.436,48.589,159.110
C00674=1023.637,171.238,-115.077,168.439,48.584,159.110
C00675=1023.644,171.521,-115.103,168.444,48.578,159.109
C00676=1023.650,171.804,-115.128,168.448,48.573,159.109
C00677=1023.656,172.086,-115.154,168.452,48.567,159.108
C00678=1023.663,172.369,-115.180,168.456,48.561,159.107
C00679=1023.668,172.618,-115.201,168.459,48.556,159.107
C00680=1023.674,172.867,-115.223,168.463,48.551,159.106
C00681=1023.680,173.116,-115.246,168.466,48.546,159.106
C00682=1023.685,173.365,-115.267,168.469,48.541,159.105
C00683=1023.691,173.614,-115.290,168.474,48.536,159.105
C00684=1023.696,173.863,-115.312,168.477,48.531,159.104
C00685=1023.703,174.112,-115.335,168.481,48.526,159.104
C00686=1023.708,174.360,-115.357,168.484,48.521,159.103
C00687=1023.713,174.609,-115.380,168.488,48.516,159.103
C00688=1023.719,174.859,-115.402,168.491,48.511,159.102
C00689=1023.725,175.107,-115.424,168.495,48.506,159.102
C00690=1023.730,175.356,-115.446,168.498,48.500,159.101
C00691=1023.736,175.605,-115.469,168.501,48.496,159.101
C00692=1023.742,175.854,-115.491,168.506,48.490,159.100
C00693=1023.748,176.103,-115.514,168.509,48.486,159.100
C00694=1023.753,176.352,-115.535,168.512,48.480,159.099
C00695=1023.759,176.601,-115.558,168.516,48.475,159.099
C00696=1023.765,176.850,-115.581,168.520,48.470,159.098
C00697=1023.770,177.099,-115.603,168.524,48.465,159.098
C00698=1023.776,177.348,-115.626,168.527,48.460,159.097
C00699=1023.782,177.597,-115.648,168.531,48.455,159.097
C00700=1023.787,177.845,-115.670,168.535,48.450,159.096
C00701=1023.793,178.094,-115.693,168.538,48.445,159.096
C00702=1023.799,178.343,-115.715,168.541,48.440,159.095
C00703=1023.805,178.592,-115.738,168.546,48.435,159.095
C00704=1023.811,178.841,-115.761,168.549,48.430,159.094
C00705=1023.816,179.091,-115.783,168.553,48.425,159.094
C00706=1023.822,179.339,-115.805,168.557,48.420,159.093
C00707=1023.828,179.588,-115.828,168.560,48.414,159.093
C00708=1023.833,179.837,-115.850,168.564,48.410,159.092
C00709=1023.839,180.086,-115.872,168.568,48.404,159.092
C00710=1023.845,180.335,-115.895,168.571,48.400,159.091
C00711=1023.851,180.584,-115.917,168.575,48.394,159.091
C00712=1023.856,180.833,-115.940,168.579,48.389,159.090
C00713=1023.863,181.082,-115.963,168.582,48.384,159.090
C00714=1023.869,181.330,-115.986,168.586,48.379,159.089
C00715=1023.874,181.580,-116.008,168.590,48.374,159.089
C00716=1023.879,181.828,-116.031,168.593,48.369,159.088
C00717=1023.886,182.077,-116.053,168.597,48.364,159.088
C00718=1023.891,182.326,-116.076,168.601,48.359,159.087
C00719=1023.897,182.575,-116.099,168.605,48.354,159.087
C00720=1023.902,182.824,-116.122,168.608,48.349,159.086
C00721=1023.908,183.073,-116.145,168.612,48.345,159.086
C00722=1023.913,183.322,-116.168,168.615,48.340,159.085
C00723=1023.918,183.571,-116.192,168.620,48.335,159.085
C00724=1023.924,183.820,-116.215,168.623,48.330,159.084
C00725=1023.930,184.069,-116.238,168.627,48.326,159.084
C00726=1023.935,184.318,-116.261,168.630,48.321,159.084
C00727=1023.941,184.567,-116.284,168.635,48.316,159.083
C00728=1023.946,184.816,-116.307,168.638,48.311,159.083
C00729=1023.951,185.064,-116.330,168.642,48.306,159.082
C00730=1023.956,185.313,-116.353,168.645,48.301,159.082
C00731=1023.963,185.561,-116.377,168.650,48.296,159.081
C00732=1023.968,185.810,-116.400,168.653,48.292,159.081
C00733=1023.973,186.059,-116.423,168.656,48.287,159.080
C00734=1023.978,186.309,-116.447,168.660,48.283,159.080
C00735=1023.984,186.557,-116.470,168.665,48.278,159.080
C00736=1023.990,186.806,-116.494,168.668,48.273,159.079
C00737=1023.995,187.055,-116.517,168.672,48.268,159.079
C00738=1024.001,187.304,-116.540,168.676,48.263,159.078
C00739=1024.007,187.586,-116.566,168.681,48.258,159.078
C00740=1024.014,187.869,-116.592,168.685,48.252,159.077
C00741=1024.019,188.151,-116.619,168.689,48.247,159.077
C00742=1024.025,188.433,-116.646,168.693,48.241,159.076
C00743=1024.031,188.681,-116.669,168.697,48.236,159.076
C00744=1024.037,188.930,-116.693,168.700,48.232,159.075
C00745=1024.042,189.179,-116.716,168.705,48.227,159.075
C00746=1024.048,189.428,-116.739,168.708,48.223,159.075
C00747=1024.053,189.677,-116.762,168.712,48.218,159.074
C00748=1024.060,189.926,-116.786,168.716,48.213,159.074
C00749=1024.065,190.175,-116.809,168.720,48.208,159.073
C00750=1024.070,190.424,-116.833,168.723,48.203,159.073
C00751=1024.076,190.672,-116.857,168.728,48.198,159.072
C00752=1024.081,190.922,-116.880,168.731,48.193,159.072
C00753=1024.087,191.170,-116.904,168.735,48.189,159.071
C00754=1024.093,191.419,-116.927,168.739,48.184,159.071
C00755=1024.098,191.668,-116.950,168.743,48.179,159.071
C00756=1024.104,191.916,-116.974,168.746,48.175,159.070
C00757=1024.110,192.165,-116.997,168.751,48.169,159.070
C00758=1024.115,192.414,-117.021,168.754,48.165,159.069
C00759=1024.121,192.663,-117.044,168.759,48.160,159.069
C00760=1024.127,192.913,-117.068,168.763,48.156,159.068
C00761=1024.133,193.161,-117.092,168.766,48.151,159.068
C00762=1024.138,193.410,-117.115,168.771,48.146,159.067
C00763=1024.144,193.658,-117.139,168.774,48.141,159.067
C00764=1024.149,193.907,-117.162,168.778,48.136,159.067
C00765=1024.155,194.156,-117.185,168.782,48.132,159.066
C00766=1024.160,194.405,-117.209,168.786,48.127,159.066
C00767=1024.167,194.654,-117.233,168.790,48.122,159.065
C00768=1024.172,194.903,-117.257,168.794,48.117,159.065
C00769=1024.178,195.151,-117.280,168.798,48.112,159.064
C00770=1024.184,195.400,-117.303,168.802,48.108,159.064
C00771=1024.189,195.649,-117.327,168.806,48.103,159.064
C00772=1024.196,195.898,-117.351,168.810,48.098,159.063
C00773=1024.201,196.147,-117.375,168.813,48.093,159.063
C00774=1024.207,196.395,-117.399,168.818,48.088,159.062
C00775=1024.212,196.644,-117.422,168.822,48.084,159.062
C00776=1024.218,196.893,-117.446,168.826,48.079,159.062
C00777=1024.224,197.142,-117.470,168.830,48.075,159.061
C00778=1024.229,197.391,-117.493,168.834,48.069,159.061
C00779=1024.235,197.639,-117.517,168.837,48.065,159.060
C00780=1024.241,197.887,-117.541,168.842,48.060,159.060
C00781=1024.247,198.137,-117.565,168.846,48.056,159.059
C00782=1024.253,198.386,-117.588,168.850,48.051,159.059
C00783=1024.258,198.634,-117.613,168.854,48.046,159.059
C00784=1024.265,198.884,-117.636,168.858,48.041,159.058
C00785=1024.271,199.132,-117.660,168.862,48.037,159.058
C00786=1024.276,199.381,-117.684,168.866,48.032,159.057
C00787=1024.282,199.629,-117.707,168.870,48.027,159.057
C00788=1024.288,199.879,-117.731,168.874,48.022,159.056
C00789=1024.294,200.127,-117.755,168.878,48.018,159.056
C00790=1024.299,200.376,-117.779,168.883,48.013,159.056
C00791=1024.305,200.625,-117.804,168.887,48.009,159.055
C00792=1024.310,200.874,-117.828,168.891,48.004,159.055
C00793=1024.315,201.122,-117.852,168.895,48.000,159.055
C00794=1024.322,201.371,-117.876,168.899,47.995,159.054
C00795=1024.327,201.620,-117.900,168.903,47.990,159.054
C00796=1024.332,201.869,-117.924,168.908,47.985,159.053
C00797=1024.338,202.118,-117.949,168.911,47.981,159.053
C00798=1024.344,202.366,-117.973,168.916,47.976,159.053
C00799=1024.350,202.615,-117.997,168.919,47.972,159.052
C00800=1024.356,202.864,-118.021,168.924,47.967,159.052
C00801=1024.361,203.113,-118.046,168.928,47.962,159.051
C00802=1024.367,203.361,-118.069,168.932,47.958,159.051
C00803=1024.390,204.394,-118.171,169.339,48.058,159.128
C00804=1024.402,204.803,-118.213,169.344,48.052,159.128
C00805=1024.412,205.213,-118.255,169.349,48.046,159.127
C00806=1024.423,205.623,-118.298,169.355,48.039,159.127
C00807=1024.433,206.033,-118.341,169.360,48.033,159.126
C00808=1024.440,206.281,-118.367,169.363,48.029,159.126
C00809=1024.447,206.531,-118.392,169.366,48.026,159.125
C00810=1024.453,206.779,-118.419,169.370,48.022,159.125
C00811=1024.459,207.027,-118.444,169.373,48.019,159.125
C00812=1024.466,207.276,-118.470,169.376,48.015,159.124
C00813=1024.473,207.525,-118.496,169.380,48.011,159.124
C00814=1024.479,207.773,-118.522,169.382,48.008,159.124
C00815=1024.486,208.021,-118.548,169.385,48.004,159.123
C00816=1024.492,208.270,-118.574,169.389,48.000,159.123
C00817=1024.498,208.518,-118.600,169.392,47.997,159.123
C00818=1024.504,208.767,-118.625,169.395,47.993,159.122
C00819=1024.512,209.016,-118.652,169.398,47.990,159.122
C00820=1024.518,209.264,-118.678,169.402,47.986,159.122
C00821=1024.524,209.513,-118.704,169.405,47.982,159.121
C00822=1024.531,209.762,-118.730,169.407,47.979,159.121
C00823=1024.537,210.010,-118.756,169.412,47.975,159.121
C00824=1024.544,210.259,-118.782,169.414,47.972,159.120
C00825=1024.550,210.507,-118.808,169.417,47.968,159.120
C00826=1024.556,210.755,-118.835,169.421,47.964,159.120
C00827=1024.563,211.004,-118.861,169.424,47.961,159.119
C00828=1024.570,211.252,-118.887,169.427,47.957,159.119
C00829=1024.575,211.501,-118.913,169.430,47.954,159.119
C00830=1024.582,211.750,-118.940,169.434,47.950,159.119
C00831=1024.588,211.998,-118.966,169.437,47.947,159.118
C00832=1024.595,212.246,-118.992,169.440,47.943,159.118
C00833=1024.602,212.495,-119.019,169.444,47.940,159.118
C00834=1024.607,212.744,-119.045,169.447,47.936,159.117
C00835=1024.614,212.993,-119.071,169.450,47.933,159.117
C00836=1024.621,213.241,-119.097,169.452,47.929,159.117
C00837=1024.627,213.489,-119.124,169.456,47.926,159.116
C00838=1024.634,213.738,-119.150,169.459,47.922,159.116
C00839=1024.640,213.986,-119.177,169.462,47.919,159.116
C00840=1024.647,214.235,-119.203,169.466,47.915,159.115
C00841=1024.653,214.483,-119.229,169.469,47.912,159.115
C00842=1024.659,214.733,-119.256,169.472,47.909,159.115
C00843=1024.666,214.981,-119.282,169.476,47.905,159.115
C00844=1024.672,215.229,-119.308,169.479,47.902,159.114
C00845=1024.679,215.478,-119.335,169.482,47.898,159.114
C00846=1024.685,215.726,-119.361,169.485,47.895,159.114
C00847=1024.692,215.975,-119.388,169.489,47.891,159.113
C00848=1024.698,216.223,-119.414,169.492,47.888,159.113
C00849=1024.705,216.472,-119.440,169.495,47.884,159.113
C00850=1024.711,216.720,-119.467,169.499,47.881,159.113
C00851=1024.718,216.969,-119.493,169.502,47.877,159.112
C00852=1024.724,217.217,-119.520,169.505,47.874,159.112
C00853=1024.731,217.466,-119.546,169.509,47.870,159.112
C00854=1024.738,217.714,-119.572,169.512,47.867,159.111
C00855=1024.744,217.963,-119.599,169.515,47.864,159.111
C00856=1024.750,218.211,-119.625,169.519,47.860,159.111
C00857=1024.757,218.460,-119.652,169.522,47.857,159.111
C00858=1024.763,218.708,-119.679,169.525,47.854,159.110
C00859=1024.770,218.957,-119.705,169.528,47.851,159.110
C00860=1024.781,219.369,-119.750,169.534,47.844,159.110
C00861=1024.791,219.782,-119.794,169.540,47.839,159.109
C00862=1024.802,220.194,-119.839,169.545,47.834,159.109
C00863=1024.812,220.607,-119.883,169.550,47.829,159.108
C00864=1024.818,220.855,-119.911,169.553,47.825,159.108
C00865=1024.826,221.104,-119.937,169.556,47.822,159.108
C00866=1024.831,221.352,-119.964,169.560,47.818,159.108
C00867=1024.838,221.601,-119.991,169.564,47.815,159.107
C00868=1024.845,221.849,-120.017,169.567,47.812,159.107
C00869=1024.851,222.098,-120.044,169.570,47.809,159.107
C00870=1024.857,222.347,-120.071,169.574,47.806,159.107
C00871=1024.864,222.594,-120.098,169.577,47.803,159.106
C00872=1024.870,222.843,-120.125,169.580,47.799,159.106
C00873=1024.876,223.092,-120.152,169.584,47.795,159.106
C00874=1024.883,223.340,-120.178,169.587,47.792,159.106
C00875=1024.889,223.588,-120.206,169.590,47.789,159.105
C00876=1024.896,223.837,-120.233,169.593,47.786,159.105
C00877=1024.903,224.086,-120.259,169.597,47.783,159.105
C00878=1024.909,224.334,-120.286,169.600,47.780,159.105
C00879=1024.915,224.583,-120.313,169.603,47.777,159.104
C00880=1024.923,224.831,-120.341,169.607,47.773,159.104
C00881=1024.929,225.079,-120.367,169.611,47.770,159.104
C00882=1024.935,225.328,-120.394,169.614,47.767,159.104
C00883=1024.942,225.577,-120.422,169.618,47.764,159.104
C00884=1024.948,225.825,-120.448,169.621,47.761,159.103
C00885=1024.955,226.073,-120.476,169.624,47.757,159.103
C00886=1024.961,226.322,-120.503,169.627,47.754,159.103
C00887=1024.968,226.570,-120.529,169.631,47.751,159.103
C00888=1024.974,226.819,-120.557,169.634,47.748,159.102
C00889=1024.981,227.068,-120.584,169.637,47.745,159.102
C00890=1024.988,227.315,-120.610,169.641,47.741,159.102
C00891=1024.994,227.564,-120.638,169.645,47.738,159.102
C00892=1025.000,227.812,-120.665,169.648,47.735,159.101
C00893=1025.007,228.061,-120.692,169.651,47.732,159.101
C00894=1025.013,228.310,-120.719,169.655,47.729,159.101
C00895=1025.020,228.558,-120.747,169.658,47.726,159.101
C00896=1025.026,228.806,-120.775,169.661,47.723,159.101
C00897=1025.032,229.055,-120.802,169.665,47.720,159.101
C00898=1025.039,229.303,-120.829,169.669,47.717,159.100
C00899=1025.045,229.552,-120.856,169.672,47.714,159.100
C00900=1025.051,229.800,-120.884,169.675,47.711,159.100
C00901=1025.058,230.049,-120.911,169.679,47.707,159.100
C00902=1025.064,230.297,-120.938,169.682,47.704,159.099
C00903=1025.071,230.545,-120.966,169.685,47.702,159.099
C00904=1025.077,230.794,-120.994,169.688,47.699,159.099
C00905=1025.084,231.042,-121.021,169.693,47.695,159.099
C00906=1025.090,231.291,-121.048,169.696,47.692,159.099
C00907=1025.096,231.539,-121.076,169.699,47.690,159.099
C00908=1025.103,231.787,-121.103,169.702,47.687,159.098
C00909=1025.110,232.036,-121.131,169.706,47.683,159.098
C00910=1025.116,232.284,-121.158,169.709,47.680,159.098
C00911=1025.122,232.533,-121.185,169.713,47.678,159.098
C00912=1025.129,232.781,-121.213,169.717,47.674,159.098
C00913=1025.136,233.030,-121.241,169.720,47.671,159.097
C00914=1025.141,233.278,-121.269,169.723,47.669,159.097
C00915=1025.148,233.526,-121.297,169.726,47.666,159.097
C00916=1025.159,233.931,-121.341,169.732,47.661,159.097
C00917=1025.169,234.335,-121.386,169.738,47.656,159.096
C00918=1025.179,234.741,-121.431,169.744,47.651,159.096
C00919=1025.189,235.145,-121.476,169.749,47.647,159.096
C00920=1025.196,235.393,-121.504,169.754,47.643,159.096
C00921=1025.203,235.641,-121.532,169.757,47.640,159.096
C00922=1025.210,235.890,-121.560,169.760,47.638,159.096
C00923=1025.216,236.138,-121.587,169.763,47.635,159.095
C00924=1025.223,236.387,-121.615,169.768,47.632,159.095
C00925=1025.230,236.635,-121.643,169.771,47.629,159.095
C00926=1025.236,236.883,-121.670,169.774,47.626,159.095
C00927=1025.242,237.132,-121.699,169.778,47.623,159.095
C00928=1025.248,237.380,-121.726,169.781,47.620,159.095
C00929=1025.255,237.629,-121.754,169.785,47.618,159.094
C00930=1025.262,237.877,-121.782,169.788,47.615,159.094
C00931=1025.268,238.125,-121.809,169.792,47.612,159.094
C00932=1025.275,238.374,-121.837,169.795,47.609,159.094
C00933=1025.281,238.623,-121.865,169.799,47.607,159.094
C00934=1025.287,238.870,-121.893,169.803,47.603,159.094
C00935=1025.294,239.119,-121.921,169.806,47.601,159.094
C00936=1025.300,239.367,-121.948,169.809,47.598,159.093
C00937=1025.307,239.615,-121.977,169.814,47.595,159.093
C00938=1025.313,239.864,-122.005,169.817,47.592,159.093
C00939=1025.320,240.112,-122.033,169.820,47.589,159.093
C00940=1025.327,240.361,-122.061,169.823,47.586,159.093
C00941=1025.333,240.609,-122.089,169.828,47.584,159.093
C00942=1025.340,240.857,-122.117,169.831,47.581,159.093
C00943=1025.346,241.106,-122.146,169.834,47.578,159.092
C00944=1025.352,241.354,-122.173,169.838,47.576,159.092
C00945=1025.358,241.602,-122.202,169.842,47.573,159.092
C00946=1025.365,241.850,-122.230,169.845,47.570,159.092
C00947=1025.371,242.099,-122.258,169.849,47.568,159.092
C00948=1025.377,242.347,-122.287,169.853,47.565,159.092
C00949=1025.384,242.595,-122.314,169.856,47.562,159.092
C00950=1025.390,242.844,-122.343,169.860,47.559,159.092
C00951=1025.397,243.092,-122.371,169.863,47.557,159.092
C00952=1025.403,243.341,-122.399,169.867,47.554,159.091
C00953=1025.410,243.589,-122.427,169.871,47.551,159.091
C00954=1025.416,243.837,-122.456,169.874,47.549,159.091
C00955=1025.423,244.086,-122.484,169.877,47.546,159.091
C00956=1025.429,244.334,-122.513,169.882,47.543,159.091
C00957=1025.435,244.583,-122.541,169.885,47.541,159.091
C00958=1025.442,244.830,-122.570,169.888,47.538,159.091
C00959=1025.448,245.079,-122.598,169.892,47.536,159.091
C00960=1025.454,245.327,-122.627,169.896,47.533,159.091
C00961=1025.461,245.575,-122.656,169.900,47.531,159.091
C00962=1025.467,245.824,-122.684,169.903,47.528,159.091
C00963=1025.473,246.072,-122.713,169.906,47.525,159.090
C00964=1025.479,246.321,-122.741,169.911,47.523,159.090
C00965=1025.486,246.569,-122.770,169.914,47.520,159.090
C00966=1025.492,246.817,-122.799,169.917,47.518,159.090
C00967=1025.498,247.065,-122.827,169.921,47.515,159.090
C00968=1025.505,247.313,-122.855,169.925,47.513,159.090
C00969=1025.512,247.561,-122.884,169.929,47.510,159.090
C00970=1025.518,247.810,-122.913,169.932,47.508,159.090
C00971=1025.524,248.058,-122.942,169.937,47.505,159.090
C00972=1025.535,248.457,-122.988,169.941,47.501,159.090
C00973=1025.544,248.855,-123.034,169.947,47.497,159.090
C00974=1025.555,249.254,-123.079,169.954,47.493,159.090
C00975=1025.565,249.652,-123.126,169.960,47.489,159.090
C00976=1025.572,249.901,-123.155,169.963,47.487,159.090
C00977=1025.579,250.148,-123.183,169.968,47.484,159.090
C00978=1025.585,250.397,-123.212,169.971,47.482,159.089
C00979=1025.591,250.645,-123.241,169.974,47.479,159.089
C00980=1025.597,250.893,-123.270,169.978,47.477,159.089
C00981=1025.604,251.141,-123.298,169.982,47.474,159.089
C00982=1025.610,251.389,-123.327,169.986,47.472,159.089
C00983=1025.617,251.638,-123.357,169.989,47.469,159.089
C00984=1025.623,251.886,-123.386,169.994,47.467,159.089
C00985=1025.630,252.135,-123.413,169.997,47.464,159.089
C00986=1025.636,252.383,-123.442,170.000,47.462,159.089
C00987=1025.643,252.631,-123.471,170.005,47.459,159.089
C00988=1025.650,252.879,-123.500,170.008,47.457,159.089
C00989=1025.656,253.128,-123.529,170.012,47.454,159.089
C00990=1025.663,253.376,-123.558,170.016,47.452,159.089
C00991=1025.669,253.624,-123.587,170.019,47.449,159.089
C00992=1025.676,253.872,-123.616,170.023,47.447,159.089
C00993=1025.682,254.120,-123.645,170.027,47.444,159.089
C00994=1025.689,254.369,-123.674,170.031,47.442,159.089
C00995=1025.695,254.617,-123.703,170.034,47.440,159.089
C00996=1025.702,254.865,-123.732,170.039,47.437,159.089
C00997=1025.708,255.113,-123.761,170.042,47.435,159.089
C00998=1025.715,255.362,-123.789,170.046,47.432,159.088
C00999=1025.722,255.610,-123.819,170.050,47.430,159.088
C01000=1025.729,255.858,-123.848,170.054,47.427,159.088
C01001=1025.735,256.106,-123.877,170.057,47.425,159.088
C01002=1025.742,256.355,-123.906,170.062,47.423,159.088
C01003=1025.748,256.603,-123.935,170.065,47.421,159.088
C01004=1025.755,256.851,-123.964,170.069,47.418,159.088
C01005=1025.762,257.099,-123.993,170.073,47.415,159.088
C01006=1025.768,257.347,-124.022,170.076,47.413,159.088
C01007=1025.774,257.596,-124.051,170.080,47.411,159.088
C01008=1025.782,257.844,-124.080,170.085,47.409,159.088
C01009=1025.788,258.092,-124.109,170.088,47.406,159.088
C01010=1025.794,258.340,-124.138,170.091,47.404,159.088
C01011=1025.801,258.589,-124.167,170.096,47.401,159.088
C01012=1025.808,258.837,-124.197,170.100,47.399,159.088
C01013=1025.815,259.085,-124.226,170.104,47.397,159.088
C01014=1025.822,259.333,-124.255,170.107,47.394,159.088
C01015=1025.828,259.582,-124.284,170.111,47.392,159.088
C01016=1025.835,259.830,-124.313,170.116,47.390,159.088
C01017=1025.842,260.078,-124.343,170.119,47.387,159.088
C01018=1025.848,260.326,-124.372,170.122,47.385,159.088
C01019=1025.855,260.575,-124.401,170.127,47.382,159.088
C01020=1025.861,260.823,-124.430,170.131,47.381,159.088
C01021=1025.868,261.070,-124.460,170.135,47.378,159.088
C01022=1025.875,261.319,-124.489,170.139,47.376,159.088
C01023=1025.881,261.567,-124.519,170.142,47.374,159.088
C01024=1025.888,261.815,-124.548,170.147,47.372,159.088
C01025=1025.894,262.063,-124.579,170.150,47.369,159.088
C01026=1025.900,262.311,-124.608,170.154,47.368,159.088
C01027=1025.907,262.560,-124.637,170.159,47.365,159.088
C01028=1025.918,262.956,-124.685,170.164,47.362,159.088
C01029=1025.928,263.353,-124.733,170.170,47.358,159.088
C01030=1025.939,263.750,-124.780,170.177,47.355,159.088
C01031=1025.949,264.147,-124.827,170.183,47.352,159.089
C01032=1025.956,264.396,-124.856,170.187,47.349,159.089
C01033=1025.961,264.644,-124.887,170.191,47.347,159.089
C01034=1025.969,264.892,-124.917,170.195,47.346,159.089
C01035=1025.975,265.140,-124.946,170.199,47.343,159.089
C01036=1025.982,265.388,-124.976,170.203,47.341,159.089
C01037=1025.988,265.636,-125.005,170.206,47.339,159.089
C01038=1025.995,265.884,-125.035,170.211,47.337,159.089
C01039=1026.001,266.132,-125.066,170.215,47.335,159.089
C01040=1026.008,266.380,-125.096,170.219,47.332,159.089
C01041=1026.015,266.629,-125.125,170.223,47.330,159.089
C01042=1026.021,266.877,-125.155,170.227,47.329,159.089
C01043=1026.028,267.125,-125.185,170.231,47.326,159.089
C01044=1026.035,267.373,-125.215,170.235,47.324,159.089
C01045=1026.040,267.621,-125.245,170.239,47.323,159.089
C01046=1026.047,267.870,-125.275,170.243,47.320,159.089
C01047=1026.054,268.117,-125.305,170.247,47.318,159.089
C01048=1026.060,268.366,-125.336,170.251,47.316,159.090
C01049=1026.067,268.614,-125.365,170.255,47.314,159.090
C01050=1026.074,268.862,-125.395,170.259,47.312,159.090
C01051=1026.080,269.110,-125.425,170.263,47.310,159.090
C01052=1026.087,269.358,-125.455,170.267,47.308,159.090
C01053=1026.093,269.605,-125.485,170.271,47.306,159.090
C01054=1026.100,269.854,-125.516,170.275,47.304,159.090
C01055=1026.106,270.101,-125.545,170.279,47.302,159.090
C01056=1026.114,270.350,-125.575,170.283,47.300,159.090
C01057=1026.120,270.598,-125.606,170.288,47.298,159.090
C01058=1026.126,270.846,-125.636,170.291,47.297,159.090
C01059=1026.133,271.094,-125.667,170.295,47.295,159.090
C01060=1026.139,271.342,-125.696,170.300,47.293,159.091
C01061=1026.146,271.590,-125.727,170.304,47.291,159.091
C01062=1026.153,271.838,-125.757,170.308,47.289,159.091
C01063=1026.159,272.086,-125.788,170.312,47.287,159.091
C01064=1026.166,272.335,-125.818,170.315,47.285,159.091
C01065=1026.172,272.582,-125.848,170.320,47.283,159.091
C01066=1026.179,272.831,-125.878,170.324,47.281,159.091
C01067=1026.185,273.079,-125.909,170.329,47.279,159.091
C01068=1026.191,273.327,-125.939,170.332,47.277,159.091
C01069=1026.199,273.574,-125.970,170.336,47.276,159.092
C01070=1026.205,273.823,-126.001,170.341,47.274,159.092
C01071=1026.212,274.071,-126.031,170.345,47.272,159.092
C01072=1026.218,274.319,-126.061,170.348,47.270,159.092
C01073=1026.225,274.568,-126.092,170.353,47.268,159.092
C01074=1026.231,274.814,-126.123,170.357,47.266,159.092
C01075=1026.238,275.063,-126.153,170.362,47.264,159.092
C01076=1026.245,275.311,-126.183,170.365,47.263,159.092
C01077=1026.251,275.559,-126.214,170.369,47.261,159.092
C01078=1026.257,275.807,-126.245,170.374,47.259,159.093
C01079=1026.265,276.055,-126.275,170.378,47.258,159.093
C01080=1026.271,276.304,-126.306,170.383,47.256,159.093
C01081=1026.278,276.551,-126.336,170.386,47.254,159.093
C01082=1026.284,276.799,-126.367,170.391,47.252,159.093
C01083=1026.291,277.048,-126.398,170.395,47.250,159.093
C01084=1026.302,277.449,-126.447,170.401,47.248,159.094
C01085=1026.312,277.851,-126.498,170.408,47.244,159.094
C01086=1026.323,278.252,-126.547,170.415,47.242,159.094
C01087=1026.334,278.654,-126.597,170.421,47.239,159.094
C01088=1026.340,278.902,-126.629,170.426,47.237,159.095
C01089=1026.346,279.149,-126.659,170.430,47.235,159.095
C01090=1026.353,279.397,-126.690,170.435,47.234,159.095
C01091=1026.360,279.646,-126.721,170.439,47.232,159.095
C01092=1026.367,279.893,-126.752,170.443,47.230,159.095
C01093=1026.374,280.141,-126.783,170.447,47.229,159.095
C01094=1026.379,280.389,-126.814,170.451,47.228,159.096
C01095=1026.386,280.637,-126.845,170.456,47.225,159.096
C01096=1026.393,280.885,-126.877,170.460,47.224,159.096
C01097=1026.399,281.134,-126.907,170.465,47.222,159.096
C01098=1026.407,281.381,-126.938,170.468,47.221,159.096
C01099=1026.413,281.629,-126.970,170.473,47.219,159.097
C01100=1026.419,281.877,-127.000,170.477,47.218,159.097
C01101=1026.426,282.125,-127.031,170.481,47.216,159.097
C01102=1026.433,282.373,-127.063,170.486,47.214,159.097
C01103=1026.439,282.621,-127.094,170.490,47.213,159.097
C01104=1026.446,282.869,-127.125,170.495,47.211,159.098
C01105=1026.453,283.117,-127.156,170.499,47.210,159.098
C01106=1026.460,283.365,-127.187,170.503,47.208,159.098
C01107=1026.466,283.613,-127.218,170.507,47.206,159.098
C01108=1026.473,283.861,-127.249,170.512,47.204,159.098
C01109=1026.480,284.109,-127.281,170.516,47.203,159.098
C01110=1026.486,284.356,-127.312,170.521,47.201,159.099
C01111=1026.493,284.604,-127.343,170.525,47.200,159.099
C01112=1026.499,284.852,-127.375,170.530,47.198,159.099
C01113=1026.507,285.100,-127.405,170.534,47.197,159.099
C01114=1026.513,285.348,-127.436,170.538,47.195,159.099
C01115=1026.520,285.596,-127.468,170.542,47.194,159.100
C01116=1026.527,285.844,-127.499,170.546,47.192,159.100
C01117=1026.534,286.092,-127.531,170.551,47.191,159.100
C01118=1026.540,286.340,-127.562,170.555,47.189,159.100
C01119=1026.547,286.588,-127.594,170.560,47.188,159.101
C01120=1026.553,286.836,-127.626,170.564,47.187,159.101
C01121=1026.560,287.084,-127.657,170.569,47.185,159.101
C01122=1026.566,287.332,-127.688,170.573,47.184,159.101
C01123=1026.573,287.579,-127.720,170.578,47.182,159.102
C01124=1026.580,287.827,-127.751,170.582,47.180,159.102
C01125=1026.587,288.075,-127.783,170.587,47.179,159.102
C01126=1026.594,288.323,-127.815,170.591,47.178,159.102
C01127=1026.600,288.570,-127.846,170.595,47.176,159.102
C01128=1026.607,288.818,-127.878,170.599,47.175,159.103
C01129=1026.613,289.067,-127.910,170.604,47.173,159.103
C01130=1026.620,289.314,-127.941,170.608,47.172,159.103
C01131=1026.627,289.562,-127.974,170.613,47.170,159.103
C01132=1026.634,289.810,-128.005,170.617,47.169,159.104
C01133=1026.641,290.058,-128.037,170.622,47.168,159.104
C01134=1026.648,290.306,-128.068,170.626,47.167,159.104
C01135=1026.654,290.554,-128.101,170.631,47.165,159.104
C01136=1026.661,290.802,-128.132,170.635,47.164,159.105
C01137=1026.667,291.050,-128.164,170.640,47.162,159.105
C01138=1026.674,291.297,-128.196,170.644,47.161,159.105
C01139=1026.681,291.545,-128.227,170.649,47.160,159.106
C01140=1026.692,291.959,-128.281,170.656,47.157,159.106
C01141=1026.704,292.373,-128.334,170.664,47.155,159.106
C01142=1026.715,292.786,-128.387,170.671,47.153,159.107
C01143=1026.726,293.201,-128.441,170.679,47.151,159.107
C01144=1026.733,293.449,-128.473,170.684,47.150,159.108
C01145=1026.740,293.696,-128.505,170.688,47.148,159.108
C01146=1026.746,293.944,-128.536,170.693,47.147,159.108
C01147=1026.753,294.191,-128.569,170.697,47.146,159.109
C01148=1026.760,294.439,-128.601,170.702,47.145,159.109
C01149=1026.766,294.687,-128.634,170.706,47.144,159.109
C01150=1026.773,294.935,-128.666,170.711,47.142,159.110
C01151=1026.780,295.182,-128.699,170.716,47.141,159.110
C01152=1026.786,295.431,-128.731,170.721,47.140,159.110
C01153=1026.792,295.678,-128.763,170.725,47.139,159.111
C01154=1026.799,295.925,-128.795,170.730,47.138,159.111
C01155=1026.806,296.174,-128.829,170.734,47.137,159.111
C01156=1026.812,296.421,-128.861,170.739,47.135,159.112
C01157=1026.819,296.669,-128.893,170.743,47.134,159.112
C01158=1026.825,296.917,-128.925,170.748,47.134,159.112
C01159=1026.832,297.165,-128.959,170.752,47.132,159.113
C01160=1026.839,297.412,-128.991,170.758,47.131,159.113
C01161=1026.845,297.660,-129.023,170.762,47.130,159.113
C01162=1026.852,297.908,-129.056,170.767,47.129,159.114
C01163=1026.859,298.156,-129.088,170.771,47.128,159.114
C01164=1026.865,298.404,-129.121,170.776,47.127,159.114
C01165=1026.872,298.651,-129.153,170.780,47.126,159.115
C01166=1026.879,298.899,-129.186,170.785,47.125,159.115
C01167=1026.886,299.147,-129.219,170.790,47.124,159.115
C01168=1026.893,299.394,-129.251,170.794,47.122,159.116
C01169=1026.899,299.642,-129.284,170.800,47.122,159.116
C01170=1026.906,299.890,-129.317,170.804,47.121,159.116
C01171=1026.913,300.137,-129.349,170.809,47.119,159.117
C01172=1026.919,300.385,-129.382,170.813,47.119,159.117
C01173=1026.926,300.633,-129.415,170.818,47.117,159.118
C01174=1026.933,300.881,-129.447,170.823,47.116,159.118
C01175=1026.940,301.129,-129.480,170.828,47.116,159.118
C01176=1026.946,301.376,-129.513,170.833,47.114,159.119
C01177=1026.953,301.624,-129.545,170.837,47.114,159.119
C01178=1026.960,301.871,-129.579,170.842,47.112,159.119
C01179=1026.967,302.119,-129.611,170.847,47.111,159.120
C01180=1026.974,302.367,-129.644,170.851,47.110,159.120
C01181=1026.981,302.615,-129.677,170.856,47.109,159.121
C01182=1026.988,302.863,-129.710,170.861,47.109,159.121
C01183=1026.995,303.110,-129.742,170.866,47.107,159.121
C01184=1027.001,303.357,-129.775,170.871,47.107,159.122
C01185=1027.008,303.605,-129.809,170.875,47.105,159.122
C01186=1027.014,303.853,-129.841,170.881,47.105,159.123
C01187=1027.022,304.101,-129.874,170.886,47.103,159.123
C01188=1027.029,304.348,-129.907,170.890,47.103,159.123
C01189=1027.036,304.596,-129.940,170.895,47.101,159.124
C01190=1027.043,304.844,-129.973,170.900,47.101,159.124
C01191=1027.049,305.092,-130.006,170.904,47.100,159.124
C01192=1027.057,305.340,-130.039,170.910,47.099,159.125
C01193=1027.064,305.587,-130.072,170.915,47.098,159.125
C01194=1027.071,305.835,-130.105,170.919,47.097,159.126
C01195=1027.077,306.082,-130.138,170.924,47.096,159.126
C01196=1027.084,306.298,-130.167,170.929,47.095,159.126
C01197=1027.089,306.513,-130.195,170.933,47.095,159.127
C01198=1027.096,306.729,-130.225,170.937,47.094,159.127
C01199=1027.102,306.944,-130.253,170.941,47.093,159.128
C01200=1027.108,307.160,-130.282,170.945,47.092,159.128
C01201=1027.114,307.376,-130.311,170.950,47.092,159.128
C01202=1027.120,307.590,-130.339,170.954,47.090,159.129
C01203=1027.126,307.806,-130.368,170.959,47.090,159.129
C01204=1027.133,308.054,-130.402,170.963,47.089,159.130
C01205=1027.141,308.301,-130.434,170.968,47.088,159.130
C01206=1027.148,308.549,-130.468,170.974,47.087,159.130
C01207=1027.155,308.797,-130.501,170.978,47.087,159.131
C01208=1027.162,309.044,-130.534,170.983,47.085,159.131
C01209=1027.169,309.292,-130.567,170.988,47.085,159.132
C01210=1027.176,309.540,-130.601,170.994,47.084,159.132
C01211=1027.183,309.788,-130.634,170.998,47.083,159.133
C01212=1027.190,310.035,-130.667,171.003,47.082,159.133
C01213=1027.198,310.282,-130.701,171.009,47.081,159.133
C01214=1027.204,310.531,-130.734,171.014,47.080,159.134
C01215=1027.212,310.777,-130.767,171.018,47.080,159.134
C01216=1027.218,311.025,-130.801,171.024,47.079,159.135
C01217=1027.225,311.273,-130.835,171.029,47.079,159.135
C01218=1027.232,311.520,-130.869,171.033,47.078,159.136
C01219=1027.238,311.768,-130.903,171.039,47.077,159.136
C01220=1027.246,312.016,-130.937,171.044,47.077,159.137
C01221=1027.253,312.263,-130.971,171.048,47.076,159.137
C01222=1027.259,312.510,-131.004,171.054,47.075,159.138
C01223=1027.266,312.758,-131.039,171.059,47.075,159.138
C01224=1027.273,313.006,-131.072,171.063,47.074,159.139
C01225=1027.280,313.253,-131.106,171.069,47.073,159.139
C01226=1027.286,313.501,-131.140,171.074,47.073,159.140
C01227=1027.293,313.749,-131.174,171.079,47.073,159.140
C01228=1027.301,313.996,-131.208,171.084,47.072,159.141
C01229=1027.306,314.243,-131.242,171.089,47.071,159.141
C01230=1027.314,314.491,-131.276,171.095,47.071,159.142
C01231=1027.321,314.738,-131.310,171.099,47.070,159.142
C01232=1027.328,314.986,-131.345,171.105,47.070,159.143
C01233=1027.335,315.234,-131.379,171.110,47.069,159.143
C01234=1027.342,315.482,-131.412,171.115,47.068,159.144
C01235=1027.348,315.729,-131.446,171.120,47.068,159.144
C01236=1027.355,315.976,-131.481,171.125,47.068,159.145
C01237=1027.363,316.224,-131.515,171.131,47.067,159.146
C01238=1027.369,316.472,-131.549,171.136,47.066,159.146
C01239=1027.376,316.719,-131.583,171.140,47.066,159.147
C01240=1027.384,316.966,-131.618,171.146,47.066,159.147
C01241=1027.390,317.214,-131.652,171.151,47.065,159.148
C01242=1027.397,317.462,-131.686,171.157,47.064,159.148
C01243=1027.405,317.709,-131.720,171.161,47.064,159.149
C01244=1027.411,317.957,-131.755,171.167,47.064,159.149
C01245=1027.419,318.205,-131.789,171.172,47.063,159.150
C01246=1027.426,318.452,-131.823,171.178,47.063,159.151
C01247=1027.433,318.700,-131.858,171.183,47.062,159.151
C01248=1027.440,318.947,-131.892,171.188,47.062,159.152
C01249=1027.447,319.195,-131.927,171.193,47.061,159.152
C01250=1027.454,319.442,-131.961,171.198,47.061,159.153
C01251=1027.461,319.689,-131.995,171.204,47.061,159.153
C01252=1027.468,319.937,-132.030,171.209,47.060,159.154
C01253=1027.475,320.184,-132.064,171.215,47.060,159.155
C01254=1027.483,320.432,-132.098,171.219,47.059,159.155
C01255=1027.489,320.680,-132.133,171.225,47.059,159.156
C01256=1027.496,320.897,-132.163,171.229,47.059,159.156
C01257=1027.502,321.115,-132.193,171.235,47.058,159.157
C01258=1027.509,321.333,-132.224,171.239,47.058,159.157
C01259=1027.514,321.551,-132.255,171.244,47.058,159.158
C01260=1027.521,321.769,-132.285,171.249,47.057,159.158
C01261=1027.528,321.987,-132.316,171.254,47.057,159.159
C01262=1027.534,322.206,-132.345,171.258,47.056,159.159
C01263=1027.540,322.424,-132.376,171.263,47.057,159.160
C01264=1027.547,322.671,-132.411,171.268,47.056,159.160
C01265=1027.555,322.918,-132.445,171.274,47.056,159.161
C01266=1027.562,323.165,-132.480,171.279,47.055,159.162
C01267=1027.569,323.414,-132.514,171.285,47.055,159.162
C01268=1027.576,323.661,-132.550,171.290,47.055,159.163
C01269=1027.584,323.908,-132.584,171.296,47.054,159.163
C01270=1027.591,324.155,-132.619,171.301,47.054,159.164
C01271=1027.598,324.403,-132.653,171.307,47.054,159.165
C01272=1027.606,324.651,-132.688,171.312,47.053,159.165
C01273=1027.612,324.898,-132.723,171.317,47.053,159.166
C01274=1027.620,325.145,-132.758,171.323,47.053,159.167
C01275=1027.628,325.393,-132.793,171.328,47.053,159.167
C01276=1027.635,325.640,-132.828,171.334,47.052,159.168
C01277=1027.642,325.887,-132.862,171.339,47.052,159.168
C01278=1027.650,326.136,-132.898,171.345,47.052,159.169
C01279=1027.657,326.383,-132.932,171.351,47.052,159.170
C01280=1027.664,326.630,-132.966,171.356,47.051,159.170
C01281=1027.672,326.878,-133.002,171.362,47.051,159.171
C01282=1027.679,327.125,-133.036,171.367,47.051,159.172
C01283=1027.686,327.373,-133.071,171.373,47.051,159.172
C01284=1027.695,327.620,-133.107,171.378,47.050,159.173
C01285=1027.701,327.867,-133.142,171.384,47.050,159.174
C01286=1027.708,328.115,-133.177,171.390,47.050,159.174
C01287=1027.715,328.363,-133.213,171.395,47.050,159.175
C01288=1027.723,328.610,-133.247,171.401,47.050,159.176
C01289=1027.730,328.856,-133.283,171.407,47.050,159.176
C01290=1027.737,329.105,-133.319,171.412,47.050,159.177
C01291=1027.744,329.352,-133.354,171.417,47.050,159.178
C01292=1027.752,329.599,-133.390,171.423,47.050,159.178
C01293=1027.759,329.847,-133.425,171.428,47.050,159.179
C01294=1027.766,330.094,-133.460,171.434,47.050,159.180
C01295=1027.774,330.341,-133.496,171.440,47.050,159.181
C01296=1027.781,330.589,-133.531,171.446,47.050,159.181
C01297=1027.788,330.836,-133.567,171.451,47.050,159.182
C01298=1027.795,331.083,-133.602,171.457,47.049,159.183
C01299=1027.803,331.331,-133.638,171.463,47.049,159.183
C01300=1027.810,331.578,-133.673,171.469,47.050,159.184
C01301=1027.818,331.825,-133.709,171.474,47.050,159.185
C01302=1027.825,332.073,-133.744,171.480,47.050,159.186
C01303=1027.832,332.320,-133.781,171.485,47.049,159.186
C01304=1027.839,332.567,-133.816,171.491,47.050,159.187
C01305=1027.847,332.815,-133.852,171.497,47.050,159.188
C01306=1027.854,333.063,-133.887,171.503,47.050,159.189
C01307=1027.862,333.309,-133.923,171.509,47.050,159.189
C01308=1027.870,333.557,-133.959,171.514,47.050,159.190
C01309=1027.876,333.804,-133.994,171.521,47.049,159.191
C01310=1027.884,334.052,-134.030,171.527,47.050,159.192
C01311=1027.891,334.298,-134.066,171.533,47.050,159.192
C01312=1027.899,334.546,-134.102,171.539,47.050,159.193
C01313=1027.906,334.794,-134.138,171.544,47.050,159.194
C01314=1027.912,335.041,-134.174,171.550,47.051,159.195
C01315=1027.920,335.288,-134.210,171.556,47.051,159.195
C01316=1027.927,335.504,-134.242,171.560,47.051,159.196
C01317=1027.933,335.720,-134.273,171.566,47.051,159.197
C01318=1027.940,335.936,-134.305,171.571,47.051,159.198
C01319=1027.946,336.151,-134.337,171.576,47.051,159.198
C01320=1027.953,336.367,-134.368,171.581,47.051,159.199
C01321=1027.959,336.583,-134.399,171.586,47.052,159.200
C01322=1027.966,336.799,-134.431,171.592,47.052,159.200
C01323=1027.972,337.014,-134.462,171.597,47.052,159.201
C01324=1027.979,337.261,-134.498,171.603,47.052,159.202
C01325=1027.986,337.509,-134.535,171.608,47.052,159.203
C01326=1027.994,337.756,-134.571,171.614,47.053,159.203
C01327=1028.002,338.003,-134.608,171.621,47.053,159.204
C01328=1028.009,338.250,-134.644,171.627,47.053,159.205
C01329=1028.017,338.497,-134.680,171.633,47.053,159.206
C01330=1028.024,338.745,-134.716,171.639,47.054,159.207
C01331=1028.032,338.992,-134.752,171.645,47.054,159.208
C01332=1028.040,339.240,-134.789,171.650,47.054,159.208
C01333=1028.046,339.487,-134.825,171.656,47.055,159.209
C01334=1028.054,339.734,-134.862,171.663,47.055,159.210
C01335=1028.062,339.981,-134.898,171.669,47.055,159.211
C01336=1028.069,340.229,-134.934,171.675,47.056,159.212
C01337=1028.077,340.476,-134.971,171.681,47.056,159.213
C01338=1028.084,340.723,-135.008,171.687,47.056,159.213
C01339=1028.092,340.971,-135.044,171.693,47.056,159.214
C01340=1028.099,341.217,-135.081,171.699,47.057,159.215
C01341=1028.106,341.464,-135.118,171.706,47.057,159.216
C01342=1028.114,341.712,-135.154,171.712,47.058,159.217
C01343=1028.122,341.959,-135.191,171.717,47.058,159.218
C01344=1028.129,342.206,-135.228,171.723,47.059,159.219
C01345=1028.137,342.453,-135.265,171.729,47.059,159.219
C01346=1028.145,342.700,-135.302,171.736,47.059,159.220
C01347=1028.152,342.948,-135.338,171.742,47.060,159.221
C01348=1028.160,343.195,-135.375,171.749,47.061,159.222
C01349=1028.167,343.442,-135.412,171.755,47.061,159.223
C01350=1028.175,343.689,-135.449,171.761,47.062,159.224
C01351=1028.183,343.936,-135.486,171.767,47.062,159.225
C01352=1028.190,344.184,-135.523,171.773,47.062,159.226
C01353=1028.198,344.431,-135.560,171.779,47.063,159.227
C01354=1028.205,344.678,-135.597,171.786,47.064,159.228
C01355=1028.213,344.925,-135.634,171.793,47.064,159.229
C01356=1028.220,345.172,-135.671,171.799,47.064,159.230
C01357=1028.228,345.419,-135.708,171.805,47.065,159.230
C01358=1028.235,345.666,-135.745,171.811,47.066,159.231
C01359=1028.243,345.913,-135.782,171.818,47.066,159.232
C01360=1028.250,346.160,-135.820,171.824,47.067,159.233
C01361=1028.258,346.407,-135.857,171.830,47.067,159.234
C01362=1028.267,346.655,-135.893,171.836,47.068,159.235
C01363=1028.274,346.902,-135.931,171.843,47.068,159.236
C01364=1028.282,347.149,-135.968,171.849,47.069,159.237
C01365=1028.289,347.396,-136.005,171.855,47.070,159.238
C01366=1028.297,347.643,-136.042,171.862,47.070,159.239
C01367=1028.304,347.890,-136.080,171.868,47.071,159.240
C01368=1028.313,348.138,-136.117,171.874,47.072,159.241
C01369=1028.320,348.385,-136.155,171.882,47.072,159.242
C01370=1028.328,348.631,-136.193,171.888,47.073,159.243
C01371=1028.336,348.878,-136.230,171.894,47.074,159.244
C01372=1028.343,349.125,-136.267,171.901,47.074,159.245
C01373=1028.351,349.373,-136.305,171.907,47.075,159.246
C01374=1028.359,349.620,-136.342,171.913,47.076,159.247
C01375=1028.366,349.867,-136.380,171.920,47.076,159.248
C01376=1028.373,350.081,-136.413,171.925,47.077,159.249
C01377=1028.380,350.295,-136.446,171.931,47.078,159.250
C01378=1028.386,350.509,-136.478,171.936,47.079,159.251
C01379=1028.393,350.723,-136.511,171.942,47.079,159.251
C01380=1028.399,350.938,-136.544,171.948,47.080,159.252
C01381=1028.406,351.152,-136.577,171.953,47.080,159.253
C01382=1028.413,351.366,-136.609,171.960,47.081,159.254
C01383=1028.420,351.581,-136.642,171.966,47.082,159.255
C01384=1028.428,351.827,-136.680,171.972,47.083,159.256
C01385=1028.435,352.074,-136.717,171.979,47.084,159.257
C01386=1028.444,352.321,-136.756,171.985,47.084,159.258
C01387=1028.451,352.568,-136.793,171.991,47.085,159.259
C01388=1028.459,352.816,-136.832,171.999,47.086,159.260
C01389=1028.467,353.062,-136.869,172.005,47.087,159.261
C01390=1028.475,353.310,-136.907,172.012,47.088,159.262
C01391=1028.483,353.556,-136.946,172.018,47.089,159.263
C01392=1028.490,353.803,-136.983,172.026,47.090,159.265
C01393=1028.499,354.050,-137.021,172.032,47.091,159.266
C01394=1028.506,354.297,-137.059,172.039,47.091,159.267
C01395=1028.514,354.545,-137.097,172.045,47.093,159.268
C01396=1028.522,354.791,-137.135,172.053,47.093,159.269
C01397=1028.531,355.038,-137.173,172.059,47.094,159.270
C01398=1028.538,355.284,-137.212,172.066,47.095,159.271
C01399=1028.546,355.532,-137.250,172.073,47.096,159.272
C01400=1028.554,355.779,-137.288,172.079,47.097,159.273
C01401=1028.562,356.026,-137.326,172.086,47.098,159.274
C01402=1028.570,356.273,-137.365,172.092,47.099,159.275
C01403=1028.577,356.520,-137.403,172.100,47.100,159.277
C01404=1028.586,356.767,-137.442,172.107,47.101,159.278
C01405=1028.593,357.013,-137.480,172.113,47.102,159.279
C01406=1028.601,357.261,-137.519,172.121,47.103,159.280
C01407=1028.609,357.508,-137.557,172.127,47.104,159.281
C01408=1028.617,357.754,-137.596,172.135,47.105,159.282
C01409=1028.625,358.002,-137.634,172.141,47.106,159.283
C01410=1028.633,358.248,-137.672,172.148,47.107,159.284
C01411=1028.641,358.495,-137.712,172.155,47.109,159.286
C01412=1028.649,358.742,-137.750,172.162,47.110,159.287
C01413=1028.658,358.989,-137.789,172.170,47.111,159.288
C01414=1028.665,359.236,-137.827,172.176,47.112,159.289
C01415=1028.673,359.483,-137.866,172.183,47.113,159.290
C01416=1028.682,359.729,-137.905,172.190,47.114,159.291
C01417=1028.689,359.976,-137.943,172.197,47.115,159.293
C01418=1028.697,360.223,-137.982,172.205,47.116,159.294
C01419=1028.706,360.470,-138.021,172.211,47.117,159.295
C01420=1028.714,360.717,-138.060,172.218,47.119,159.296
C01421=1028.722,360.964,-138.099,172.225,47.120,159.297
C01422=1028.730,361.210,-138.138,172.232,47.121,159.299
C01423=1028.738,361.457,-138.177,172.240,47.123,159.300
C01424=1028.746,361.704,-138.216,172.246,47.124,159.301
C01425=1028.754,361.951,-138.255,172.254,47.125,159.302
C01426=1028.762,362.197,-138.294,172.261,47.126,159.304
C01427=1028.770,362.444,-138.334,172.268,47.128,159.305
C01428=1028.778,362.691,-138.373,172.276,47.129,159.306
C01429=1028.786,362.937,-138.412,172.283,47.130,159.307
C01430=1028.795,363.185,-138.451,172.289,47.132,159.308
C01431=1028.802,363.432,-138.491,172.297,47.133,159.310
C01432=1028.811,363.678,-138.530,172.305,47.134,159.311
C01433=1028.819,363.925,-138.569,172.311,47.136,159.312
C01434=1028.827,364.172,-138.608,172.319,47.137,159.314
C01435=1028.835,364.419,-138.648,172.326,47.139,159.315
C01436=1028.842,364.636,-138.683,172.333,47.140,159.316
C01437=1028.849,364.854,-138.717,172.339,47.141,159.317
C01438=1028.857,365.071,-138.752,172.345,47.142,159.318
C01439=1028.864,365.288,-138.787,172.352,47.143,159.319
C01440=1028.871,365.506,-138.822,172.358,47.145,159.321
C01441=1028.878,365.723,-138.856,172.365,47.146,159.322
C01442=1028.886,365.940,-138.891,172.371,47.148,159.323
C01443=1028.893,366.157,-138.926,172.378,47.148,159.324
C01444=1028.901,366.404,-138.966,172.385,47.150,159.325
C01445=1028.910,366.651,-139.005,172.393,47.151,159.327
C01446=1028.918,366.897,-139.044,172.400,47.153,159.328
C01447=1028.926,367.145,-139.085,172.408,47.154,159.329
C01448=1028.935,367.391,-139.124,172.416,47.156,159.331
C01449=1028.943,367.638,-139.163,172.422,47.157,159.332
C01450=1028.951,367.884,-139.204,172.430,47.159,159.333
C01451=1028.960,368.131,-139.243,172.438,47.161,159.335
C01452=1028.968,368.377,-139.283,172.445,47.162,159.336
C01453=1028.977,368.625,-139.322,172.453,47.163,159.337
C01454=1028.985,368.871,-139.363,172.461,47.165,159.339
C01455=1028.994,369.118,-139.402,172.468,47.167,159.340
C01456=1029.002,369.365,-139.442,172.476,47.168,159.341
C01457=1029.011,369.611,-139.483,172.483,47.170,159.343
C01458=1029.019,369.858,-139.522,172.491,47.171,159.344
C01459=1029.027,370.104,-139.563,172.498,47.173,159.346
C01460=1029.035,370.350,-139.603,172.506,47.175,159.347
C01461=1029.043,370.597,-139.643,172.514,47.177,159.348
C01462=1029.052,370.844,-139.683,172.522,47.179,159.350
C01463=1029.060,371.091,-139.723,172.529,47.180,159.351
C01464=1029.068,371.337,-139.764,172.537,47.182,159.353
C01465=1029.078,371.584,-139.804,172.545,47.183,159.354
C01466=1029.086,371.830,-139.845,172.553,47.185,159.356
C01467=1029.093,372.077,-139.885,172.561,47.187,159.357
C01468=1029.103,372.324,-139.925,172.569,47.189,159.359
C01469=1029.111,372.570,-139.966,172.576,47.190,159.360
C01470=1029.119,372.816,-140.007,172.584,47.192,159.361
C01471=1029.128,373.063,-140.047,172.592,47.194,159.363
C01472=1029.136,373.309,-140.088,172.600,47.196,159.364
C01473=1029.146,373.556,-140.128,172.608,47.198,159.366
C01474=1029.154,373.802,-140.169,172.616,47.200,159.367
C01475=1029.162,374.049,-140.210,172.623,47.201,159.369
C01476=1029.171,374.295,-140.250,172.631,47.203,159.370
C01477=1029.180,374.542,-140.291,172.639,47.205,159.372
C01478=1029.188,374.788,-140.331,172.647,47.207,159.373
C01479=1029.197,375.035,-140.372,172.655,47.209,159.375
C01480=1029.205,375.281,-140.412,172.663,47.210,159.376
C01481=1029.214,375.528,-140.453,172.671,47.212,159.378
C01482=1029.222,375.774,-140.493,172.679,47.214,159.379
C01483=1029.231,376.021,-140.534,172.688,47.216,159.381
C01484=1029.240,376.268,-140.576,172.696,47.218,159.382
C01485=1029.249,376.514,-140.616,172.704,47.220,159.384
C01486=1029.257,376.761,-140.657,172.712,47.222,159.385
C01487=1029.267,377.007,-140.698,172.720,47.224,159.387
C01488=1029.275,377.253,-140.739,172.728,47.226,159.388
C01489=1029.284,377.500,-140.780,172.736,47.228,159.390
C01490=1029.293,377.746,-140.822,172.745,47.230,159.392
C01491=1029.301,377.993,-140.862,172.753,47.232,159.393
C01492=1029.310,378.239,-140.904,172.761,47.234,159.395
C01493=1029.318,378.486,-140.945,172.769,47.236,159.396
C01494=1029.327,378.732,-140.986,172.777,47.239,159.398
C01495=1029.335,378.978,-141.028,172.786,47.240,159.400
C01496=1029.343,379.206,-141.067,172.793,47.242,159.401
C01497=1029.351,379.434,-141.105,172.801,47.244,159.403
C01498=1029.360,379.662,-141.142,172.809,47.246,159.404
C01499=1029.368,379.890,-141.181,172.817,47.249,159.406
C01500=1029.376,380.118,-141.220,172.824,47.251,159.407
C01501=1029.384,380.346,-141.258,172.832,47.253,159.409
C01502=1029.392,380.574,-141.297,172.840,47.255,159.410
C01503=1029.400,380.801,-141.335,172.848,47.256,159.412
C01504=1029.409,381.048,-141.376,172.856,47.259,159.413
C01505=1029.418,381.294,-141.418,172.864,47.261,159.415
C01506=1029.427,381.540,-141.460,172.873,47.263,159.417
C01507=1029.436,381.787,-141.501,172.881,47.265,159.418
C01508=1029.445,382.033,-141.543,172.890,47.268,159.420
C01509=1029.454,382.280,-141.585,172.899,47.270,159.422
C01510=1029.463,382.526,-141.627,172.907,47.272,159.424
C01511=1029.472,382.772,-141.668,172.916,47.275,159.425
C01512=1029.481,383.019,-141.710,172.924,47.277,159.427
C01513=1029.490,383.264,-141.752,172.933,47.280,159.429
C01514=1029.499,383.511,-141.794,172.942,47.282,159.430
C01515=1029.508,383.757,-141.836,172.950,47.284,159.432
C01516=1029.517,384.004,-141.878,172.959,47.286,159.434
C01517=1029.526,384.249,-141.920,172.968,47.289,159.436
C01518=1029.535,384.496,-141.962,172.976,47.291,159.437
C01519=1029.544,384.742,-142.003,172.985,47.293,159.439
C01520=1029.553,384.988,-142.046,172.993,47.296,159.441
C01521=1029.563,385.235,-142.088,173.003,47.298,159.443
C01522=1029.571,385.481,-142.130,173.011,47.300,159.444
C01523=1029.580,385.727,-142.173,173.020,47.303,159.446
C01524=1029.589,385.974,-142.214,173.029,47.306,159.448
C01525=1029.599,386.220,-142.257,173.038,47.308,159.450
C01526=1029.608,386.466,-142.300,173.048,47.310,159.452
C01527=1029.617,386.712,-142.341,173.056,47.313,159.453
C01528=1029.626,386.958,-142.384,173.065,47.315,159.455
C01529=1029.636,387.204,-142.427,173.074,47.318,159.457
C01530=1029.645,387.451,-142.468,173.083,47.320,159.459
C01531=1029.654,387.697,-142.511,173.091,47.323,159.461
C01532=1029.663,387.942,-142.554,173.101,47.325,159.462
C01533=1029.673,388.189,-142.597,173.110,47.328,159.464
C01534=1029.681,388.435,-142.640,173.119,47.331,159.466
C01535=1029.690,388.681,-142.682,173.128,47.333,159.468
C01536=1029.700,388.927,-142.725,173.137,47.336,159.470
C01537=1029.709,389.173,-142.767,173.146,47.339,159.472
C01538=1029.719,389.420,-142.811,173.155,47.341,159.474
C01539=1029.728,389.665,-142.853,173.164,47.344,159.476
C01540=1029.737,389.911,-142.895,173.174,47.347,159.477
C01541=1029.746,390.158,-142.939,173.183,47.349,159.479
C01542=1029.755,390.404,-142.981,173.192,47.352,159.481
C01543=1029.765,390.650,-143.025,173.201,47.355,159.483
C01544=1029.774,390.896,-143.068,173.211,47.358,159.485
C01545=1029.784,391.142,-143.111,173.220,47.360,159.487
C01546=1029.793,391.387,-143.154,173.229,47.363,159.489
C01547=1029.803,391.634,-143.197,173.239,47.366,159.491
C01548=1029.811,391.880,-143.240,173.248,47.369,159.493
C01549=1029.821,392.126,-143.284,173.258,47.371,159.495
C01550=1029.830,392.372,-143.327,173.267,47.374,159.497
C01551=1029.840,392.618,-143.370,173.276,47.377,159.499
C01552=1029.850,392.864,-143.413,173.286,47.380,159.501
C01553=1029.858,393.109,-143.457,173.295,47.383,159.503
C01554=1029.869,393.355,-143.500,173.305,47.386,159.505
C01555=1029.878,393.602,-143.544,173.315,47.388,159.507
C01556=1029.887,393.847,-143.587,173.324,47.392,159.509
C01557=1029.897,394.093,-143.631,173.333,47.395,159.511
C01558=1029.906,394.338,-143.674,173.343,47.398,159.513
C01559=1029.916,394.585,-143.718,173.353,47.401,159.515
C01560=1029.926,394.830,-143.762,173.362,47.403,159.517
C01561=1029.935,395.076,-143.805,173.372,47.407,159.519
C01562=1029.945,395.322,-143.849,173.382,47.410,159.521
C01563=1029.954,395.568,-143.893,173.392,47.412,159.523
C01564=1029.963,395.813,-143.937,173.401,47.416,159.526
C01565=1029.973,396.059,-143.980,173.411,47.419,159.528
C01566=1029.982,396.305,-144.024,173.421,47.422,159.530
C01567=1029.992,396.551,-144.069,173.431,47.425,159.532
C01568=1030.002,396.797,-144.112,173.441,47.428,159.534
C01569=1030.011,397.043,-144.156,173.451,47.431,159.536
C01570=1030.022,397.288,-144.200,173.460,47.434,159.538
C01571=1030.031,397.535,-144.245,173.470,47.437,159.540
C01572=1030.041,397.781,-144.289,173.480,47.440,159.542
C01573=1030.051,398.026,-144.333,173.490,47.444,159.545
C01574=1030.061,398.272,-144.377,173.500,47.447,159.547
C01575=1030.070,398.518,-144.421,173.511,47.450,159.549
C01576=1030.080,398.763,-144.465,173.521,47.453,159.551
C01577=1030.090,399.010,-144.509,173.531,47.456,159.553
C01578=1030.100,399.255,-144.554,173.541,47.459,159.555
C01579=1030.109,399.501,-144.598,173.551,47.463,159.558
C01580=1030.119,399.746,-144.643,173.561,47.466,159.560
C01581=1030.129,399.992,-144.687,173.571,47.470,159.562
C01582=1030.139,400.239,-144.732,173.582,47.473,159.564
C01583=1030.149,400.484,-144.777,173.592,47.476,159.567
C01584=1030.159,400.730,-144.822,173.602,47.480,159.569
C01585=1030.168,400.975,-144.866,173.612,47.483,159.571
C01586=1030.179,401.220,-144.911,173.623,47.486,159.574
C01587=1030.189,401.467,-144.955,173.633,47.490,159.576
C01588=1030.199,401.713,-145.000,173.643,47.493,159.578
C01589=1030.208,401.958,-145.045,173.654,47.497,159.581
C01590=1030.218,402.204,-145.090,173.664,47.500,159.583
C01591=1030.228,402.450,-145.135,173.675,47.504,159.585
C01592=1030.238,402.695,-145.180,173.685,47.507,159.587
C01593=1030.248,402.940,-145.225,173.696,47.510,159.590
C01594=1030.258,403.187,-145.270,173.706,47.514,159.592
C01595=1030.268,403.432,-145.315,173.717,47.518,159.594
C01596=1030.279,403.678,-145.361,173.727,47.521,159.597
C01597=1030.288,403.923,-145.406,173.738,47.525,159.599
C01598=1030.297,404.169,-145.451,173.749,47.528,159.602
C01599=1030.308,404.415,-145.497,173.759,47.532,159.604
C01600=1030.318,404.660,-145.542,173.771,47.536,159.606
C01601=1030.328,404.906,-145.587,173.781,47.539,159.609
C01602=1030.339,405.152,-145.633,173.792,47.543,159.611
C01603=1030.349,405.397,-145.679,173.802,47.547,159.614
C01604=1030.359,405.643,-145.724,173.814,47.550,159.616
C01605=1030.369,405.888,-145.769,173.824,47.554,159.618
C01606=1030.379,406.134,-145.815,173.835,47.558,159.621
C01607=1030.390,406.380,-145.860,173.846,47.562,159.623
C01608=1030.400,406.625,-145.906,173.857,47.565,159.626
C01609=1030.410,406.871,-145.951,173.868,47.568,159.628
C01610=1030.421,407.117,-145.997,173.879,47.573,159.631
C01611=1030.431,407.361,-146.043,173.890,47.576,159.633
C01612=1030.441,407.607,-146.089,173.901,47.580,159.636
C01613=1030.451,407.853,-146.135,173.912,47.584,159.638
C01614=1030.462,408.099,-146.181,173.924,47.588,159.641
C01615=1030.473,408.344,-146.227,173.935,47.591,159.643
C01616=1030.484,408.611,-146.277,173.947,47.596,159.646
C01617=1030.495,408.878,-146.326,173.959,47.600,159.649
C01618=1030.507,409.146,-146.377,173.971,47.604,159.652
C01619=1030.519,409.412,-146.427,173.983,47.608,159.655
C01620=1030.529,409.658,-146.473,173.995,47.612,159.657
C01621=1030.540,409.903,-146.518,174.006,47.616,159.660
C01622=1030.551,410.149,-146.564,174.018,47.620,159.662
C01623=1030.561,410.394,-146.612,174.029,47.624,159.665
C01624=1030.571,410.640,-146.658,174.041,47.628,159.668
C01625=1030.582,410.885,-146.704,174.052,47.633,159.670
C01626=1030.592,411.131,-146.751,174.064,47.636,159.673
C01627=1030.603,411.376,-146.797,174.075,47.640,159.676
C01628=1030.613,411.622,-146.844,174.087,47.644,159.678
C01629=1030.624,411.866,-146.890,174.098,47.648,159.681
C01630=1030.635,412.111,-146.937,174.110,47.653,159.684
C01631=1030.646,412.357,-146.985,174.122,47.657,159.687
C01632=1030.656,412.603,-147.030,174.134,47.661,159.689
C01633=1030.667,412.848,-147.078,174.145,47.665,159.692
C01634=1030.677,413.093,-147.124,174.157,47.669,159.695
C01635=1030.689,413.339,-147.171,174.169,47.674,159.698
C01636=1030.699,413.584,-147.219,174.181,47.677,159.700
C01637=1030.710,413.829,-147.265,174.193,47.682,159.703
C01638=1030.721,414.075,-147.313,174.205,47.686,159.706
C01639=1030.732,414.320,-147.359,174.217,47.690,159.709
C01640=1030.742,414.565,-147.407,174.229,47.694,159.711
C01641=1030.754,414.811,-147.454,174.241,47.699,159.714
C01642=1030.764,415.056,-147.500,174.253,47.703,159.717
C01643=1030.776,415.301,-147.548,174.265,47.708,159.720
C01644=1030.786,415.546,-147.595,174.278,47.712,159.723
C01645=1030.797,415.792,-147.643,174.290,47.716,159.726
C01646=1030.809,416.037,-147.690,174.302,47.720,159.728
C01647=1030.819,416.283,-147.738,174.314,47.725,159.732
C01648=1030.830,416.528,-147.784,174.327,47.730,159.734
C01649=1030.841,416.773,-147.833,174.339,47.734,159.737
C01650=1030.853,417.018,-147.880,174.351,47.738,159.740
C01651=1030.863,417.263,-147.927,174.364,47.742,159.743
C01652=1030.874,417.509,-147.976,174.376,47.748,159.746
C01653=1030.886,417.754,-148.023,174.388,47.752,159.749
C01654=1030.896,417.999,-148.071,174.401,47.757,159.752
C01655=1030.908,418.245,-148.119,174.413,47.761,159.755
C01656=1030.919,418.490,-148.167,174.427,47.766,159.758
C01657=1030.930,418.734,-148.215,174.439,47.770,159.761
C01658=1030.941,418.980,-148.263,174.452,47.775,159.764
C01659=1030.952,419.225,-148.311,174.464,47.780,159.767
C01660=1030.964,419.470,-148.359,174.477,47.784,159.770
C01661=1030.975,419.715,-148.407,174.490,47.789,159.773
C01662=1030.986,419.961,-148.455,174.503,47.793,159.776
C01663=1030.998,420.204,-148.504,174.516,47.798,159.779
C01664=1031.009,420.450,-148.552,174.529,47.803,159.783
C01665=1031.020,420.695,-148.600,174.542,47.808,159.786
C01666=1031.032,420.940,-148.648,174.555,47.812,159.789
C01667=1031.043,421.185,-148.697,174.568,47.817,159.792
C01668=1031.054,421.430,-148.745,174.581,47.822,159.795
C01669=1031.066,421.676,-148.795,174.594,47.827,159.798
C01670=1031.078,421.921,-148.842,174.608,47.831,159.801
C01671=1031.089,422.166,-148.891,174.620,47.837,159.805
C01672=1031.101,422.411,-148.940,174.634,47.841,159.808
C01673=1031.113,422.655,-148.988,174.647,47.846,159.811
C01674=1031.124,422.900,-149.037,174.661,47.851,159.814
C01675=1031.136,423.146,-149.086,174.674,47.856,159.817
C01676=1031.149,423.423,-149.141,174.689,47.862,159.821
C01677=1031.162,423.700,-149.197,174.704,47.867,159.825
C01678=1031.175,423.977,-149.253,174.720,47.873,159.829
C01679=1031.189,424.254,-149.308,174.735,47.878,159.832
C01680=1031.200,424.499,-149.357,174.748,47.883,159.836
C01681=1031.212,424.744,-149.406,174.762,47.889,159.839
C01682=1031.224,424.989,-149.455,174.776,47.894,159.842
C01683=1031.235,425.234,-149.504,174.790,47.899,159.846
C01684=1031.247,425.478,-149.554,174.804,47.904,159.849
C01685=1031.259,425.724,-149.604,174.818,47.909,159.852
C01686=1031.270,425.968,-149.653,174.831,47.914,159.856
C01687=1031.282,426.213,-149.703,174.845,47.920,159.859
C01688=1031.294,426.459,-149.752,174.859,47.925,159.863
C01689=1031.306,426.703,-149.802,174.874,47.929,159.866
C01690=1031.318,426.948,-149.851,174.888,47.935,159.870
C01691=1031.330,427.192,-149.901,174.902,47.940,159.873
C01692=1031.342,427.437,-149.951,174.916,47.946,159.877
C01693=1031.354,427.683,-150.000,174.930,47.951,159.880
C01694=1031.366,427.927,-150.050,174.944,47.956,159.884
C01695=1031.378,428.172,-150.101,174.958,47.962,159.887
C01696=1031.390,428.417,-150.151,174.973,47.967,159.891
C01697=1031.402,428.661,-150.201,174.987,47.972,159.894
C01698=1031.414,428.906,-150.251,175.002,47.977,159.898
C01699=1031.426,429.150,-150.301,175.016,47.983,159.901
C01700=1031.438,429.395,-150.351,175.031,47.988,159.905
C01701=1031.450,429.640,-150.402,175.045,47.994,159.908
C01702=1031.463,429.885,-150.452,175.060,47.999,159.912
C01703=1031.474,430.129,-150.502,175.074,48.005,159.916
C01704=1031.487,430.373,-150.553,175.090,48.011,159.920
C01705=1031.499,430.618,-150.603,175.105,48.016,159.923
C01706=1031.512,430.863,-150.653,175.119,48.021,159.927
C01707=1031.524,431.107,-150.704,175.134,48.027,159.931
C01708=1031.536,431.351,-150.755,175.149,48.032,159.934
C01709=1031.549,431.597,-150.806,175.165,48.038,159.938
C01710=1031.562,431.841,-150.857,175.179,48.044,159.942
C01711=1031.574,432.085,-150.907,175.194,48.050,159.946
C01712=1031.587,432.330,-150.957,175.210,48.055,159.949
C01713=1031.598,432.574,-151.009,175.225,48.061,159.953
C01714=1031.611,432.819,-151.060,175.240,48.066,159.957
C01715=1031.624,433.064,-151.111,175.256,48.072,159.961
C01716=1031.637,433.308,-151.162,175.271,48.078,159.965
C01717=1031.650,433.552,-151.212,175.286,48.084,159.968
C01718=1031.662,433.797,-151.264,175.302,48.089,159.972
C01719=1031.675,434.041,-151.315,175.318,48.096,159.976
C01720=1031.688,434.286,-151.366,175.333,48.101,159.980
C01721=1031.700,434.530,-151.418,175.349,48.107,159.984
C01722=1031.713,434.774,-151.469,175.364,48.113,159.988
C01723=1031.726,435.019,-151.521,175.380,48.119,159.992
C01724=1031.738,435.263,-151.572,175.396,48.124,159.996
C01725=1031.752,435.507,-151.624,175.412,48.131,160.000
C01726=1031.764,435.752,-151.675,175.428,48.137,160.004
C01727=1031.777,435.996,-151.728,175.443,48.142,160.008
C01728=1031.791,436.241,-151.780,175.460,48.148,160.012
C01729=1031.802,436.485,-151.831,175.476,48.155,160.016
C01730=1031.816,436.729,-151.883,175.492,48.161,160.020
C01731=1031.828,436.973,-151.935,175.508,48.167,160.024
C01732=1031.842,437.217,-151.987,175.524,48.173,160.028
C01733=1031.854,437.462,-152.039,175.541,48.179,160.033
C01734=1031.868,437.706,-152.091,175.557,48.185,160.037
C01735=1031.881,437.950,-152.143,175.574,48.191,160.041
C01736=1031.896,438.239,-152.205,175.593,48.199,160.046
C01737=1031.912,438.528,-152.268,175.613,48.206,160.051
C01738=1031.928,438.817,-152.330,175.633,48.213,160.056
C01739=1031.943,439.107,-152.391,175.652,48.221,160.061
C01740=1031.956,439.337,-152.441,175.668,48.227,160.065
C01741=1031.968,439.567,-152.491,175.685,48.232,160.069
C01742=1031.981,439.798,-152.541,175.700,48.238,160.073
C01743=1031.993,440.027,-152.590,175.716,48.245,160.077
C01744=1032.006,440.258,-152.640,175.732,48.251,160.081
C01745=1032.019,440.488,-152.690,175.748,48.257,160.085
C01746=1032.031,440.718,-152.740,175.765,48.263,160.090
C01747=1032.044,440.948,-152.790,175.781,48.269,160.094
C01748=1032.058,441.192,-152.843,175.798,48.275,160.098
C01749=1032.071,441.436,-152.896,175.815,48.282,160.103
C01750=1032.085,441.679,-152.948,175.832,48.288,160.107
C01751=1032.099,441.924,-153.002,175.850,48.295,160.112
C01752=1032.112,442.168,-153.055,175.867,48.301,160.116
C01753=1032.126,442.411,-153.109,175.886,48.308,160.120
C01754=1032.140,442.656,-153.162,175.903,48.314,160.125
C01755=1032.153,442.899,-153.215,175.920,48.321,160.129
C01756=1032.167,443.142,-153.268,175.938,48.328,160.134
C01757=1032.181,443.386,-153.322,175.957,48.334,160.139
C01758=1032.195,443.629,-153.375,175.974,48.341,160.143
C01759=1032.210,443.873,-153.428,175.992,48.348,160.148
C01760=1032.225,444.115,-153.480,176.010,48.353,160.152
C01761=1032.240,444.358,-153.532,176.028,48.360,160.157
C01762=1032.256,444.602,-153.584,176.046,48.367,160.162
C01763=1032.273,444.847,-153.634,176.064,48.372,160.166
C01764=1032.291,445.090,-153.685,176.083,48.379,160.171
C01765=1032.308,445.333,-153.736,176.102,48.384,160.175
C01766=1032.326,445.577,-153.785,176.120,48.391,160.180
C01767=1032.345,445.821,-153.835,176.138,48.396,160.184
C01768=1032.364,446.066,-153.883,176.158,48.402,160.189
C01769=1032.384,446.309,-153.932,176.176,48.408,160.193
C01770=1032.404,446.554,-153.980,176.195,48.413,160.197
C01771=1032.424,446.799,-154.028,176.214,48.419,160.202
C01772=1032.445,447.042,-154.075,176.233,48.425,160.206
C01773=1032.467,447.287,-154.122,176.252,48.430,160.211
C01774=1032.489,447.532,-154.169,176.271,48.435,160.215
C01775=1032.512,447.777,-154.215,176.291,48.440,160.220
C01776=1032.535,448.020,-154.260,176.310,48.445,160.224
C01777=1032.558,448.265,-154.306,176.329,48.451,160.229
C01778=1032.582,448.511,-154.350,176.349,48.456,160.233
C01779=1032.608,448.756,-154.394,176.368,48.461,160.238
C01780=1032.633,449.000,-154.439,176.388,48.465,160.242
C01781=1032.658,449.245,-154.483,176.408,48.470,160.246
C01782=1032.685,449.490,-154.525,176.428,48.475,160.251
C01783=1032.711,449.735,-154.568,176.448,48.480,160.255
C01784=1032.738,449.980,-154.610,176.468,48.484,160.259
